C01827=1172.845,288.694,-69.686,-176.933,7.790,148.605
C01828=1172.841,288.942,-69.715,-176.930,7.793,148.605
C01829=1172.837,289.190,-69.744,-176.927,7.796,148.605
C01830=1172.832,289.439,-69.774,-176.925,7.799,148.605
C01831=1172.828,289.687,-69.805,-176.922,7.802,148.605
C01832=1172.824,289.935,-69.834,-176.920,7.805,148.605
C01833=1172.819,290.183,-69.864,-176.917,7.808,148.605
C01834=1172.815,290.431,-69.893,-176.914,7.811,148.605
C01835=1172.811,290.680,-69.923,-176.912,7.814,148.605
C01836=1172.807,290.928,-69.952,-176.910,7.816,148.605
C01837=1172.803,291.176,-69.981,-176.907,7.819,148.605
C01838=1172.798,291.424,-70.012,-176.904,7.822,148.605
C01839=1172.794,291.673,-70.042,-176.901,7.825,148.605
C01840=1172.790,291.921,-70.071,-176.899,7.828,148.605
C01841=1172.785,292.169,-70.101,-176.896,7.831,148.605
C01842=1172.781,292.417,-70.131,-176.894,7.834,148.605
C01843=1172.777,292.665,-70.161,-176.891,7.837,148.605
C01844=1172.772,292.914,-70.190,-176.889,7.841,148.605
C01845=1172.768,293.162,-70.220,-176.886,7.844,148.605
C01846=1172.764,293.409,-70.250,-176.883,7.847,148.605
C01847=1172.760,293.658,-70.280,-176.881,7.849,148.605
C01848=1172.755,293.906,-70.309,-176.878,7.852,148.605
C01849=1172.751,294.154,-70.339,-176.876,7.855,148.605
C01850=1172.747,294.403,-70.370,-176.873,7.858,148.605
C01851=1172.742,294.651,-70.399,-176.871,7.861,148.605
C01852=1172.738,294.898,-70.429,-176.868,7.864,148.605
C01853=1172.734,295.147,-70.459,-176.866,7.867,148.605
C01854=1172.730,295.395,-70.489,-176.863,7.870,148.605
C01855=1172.726,295.643,-70.519,-176.860,7.873,148.605
C01856=1172.721,295.891,-70.548,-176.857,7.876,148.605
C01857=1172.717,296.140,-70.579,-176.855,7.880,148.605
C01858=1172.713,296.388,-70.609,-176.852,7.883,148.605
C01859=1172.709,296.636,-70.640,-176.850,7.886,148.605
C01860=1172.704,296.884,-70.669,-176.847,7.888,148.605
C01861=1172.700,297.132,-70.699,-176.845,7.891,148.605
C01862=1172.696,297.381,-70.729,-176.842,7.894,148.605
C01863=1172.692,297.628,-70.759,-176.840,7.897,148.605
C01864=1172.687,297.876,-70.789,-176.837,7.900,148.605
C01865=1172.683,298.124,-70.820,-176.835,7.903,148.605
C01866=1172.679,298.373,-70.849,-176.832,7.906,148.605
C01867=1172.675,298.621,-70.880,-176.829,7.909,148.605
C01868=1172.671,298.869,-70.910,-176.827,7.912,148.606
C01869=1172.666,299.118,-70.940,-176.824,7.915,148.606
C01870=1172.662,299.365,-70.971,-176.821,7.918,148.606
C01871=1172.657,299.614,-71.001,-176.819,7.921,148.605
C01872=1172.653,299.861,-71.031,-176.816,7.925,148.606
C01873=1172.649,300.110,-71.062,-176.814,7.928,148.606
C01874=1172.645,300.358,-71.091,-176.811,7.931,148.606
C01875=1172.640,300.606,-71.122,-176.809,7.934,148.606
C01876=1172.637,300.854,-71.152,-176.806,7.937,148.606
C01877=1172.632,301.102,-71.183,-176.804,7.939,148.606
C01878=1172.628,301.350,-71.213,-176.801,7.942,148.606
C01879=1172.624,301.599,-71.244,-176.799,7.945,148.606
C01880=1172.620,301.847,-71.274,-176.796,7.948,148.606
C01881=1172.615,302.094,-71.305,-176.793,7.951,148.606
C01882=1172.611,302.343,-71.334,-176.791,7.955,148.606
C01883=1172.606,302.591,-71.365,-176.788,7.958,148.606
C01884=1172.602,302.839,-71.396,-176.786,7.961,148.606
C01885=1172.599,303.087,-71.426,-176.783,7.964,148.606
C01886=1172.594,303.335,-71.457,-176.781,7.967,148.606
C01887=1172.590,303.583,-71.486,-176.778,7.970,148.606
C01888=1172.586,303.832,-71.518,-176.776,7.973,148.606
C01889=1172.581,304.080,-71.548,-176.773,7.976,148.606
C01890=1172.577,304.328,-71.578,-176.770,7.979,148.606
C01891=1172.573,304.575,-71.609,-176.768,7.982,148.606
C01892=1172.568,304.823,-71.640,-176.765,7.985,148.606
C01893=1172.565,305.072,-71.671,-176.763,7.989,148.607
C01894=1172.560,305.320,-71.701,-176.760,7.992,148.607
C01895=1172.556,305.568,-71.732,-176.757,7.995,148.607
C01896=1172.552,305.816,-71.763,-176.755,7.998,148.607
C01897=1172.547,306.065,-71.793,-176.752,8.001,148.607
C01898=1172.543,306.313,-71.823,-176.750,8.004,148.607
C01899=1172.539,306.560,-71.854,-176.747,8.007,148.607
C01900=1172.535,306.809,-71.885,-176.745,8.010,148.607
C01901=1172.531,307.056,-71.916,-176.742,8.013,148.607
C01902=1172.526,307.304,-71.947,-176.739,8.017,148.607
C01903=1172.523,307.553,-71.977,-176.737,8.019,148.607
C01904=1172.518,307.800,-72.008,-176.734,8.023,148.607
C01905=1172.513,308.048,-72.039,-176.732,8.026,148.607
C01906=1172.509,308.297,-72.070,-176.729,8.029,148.607
C01907=1172.505,308.545,-72.101,-176.727,8.032,148.607
C01908=1172.501,308.793,-72.131,-176.724,8.035,148.607
C01909=1172.497,309.041,-72.162,-176.721,8.038,148.607
C01910=1172.492,309.289,-72.193,-176.719,8.041,148.608
C01911=1172.488,309.537,-72.224,-176.716,8.044,148.607
C01912=1172.484,309.785,-72.256,-176.714,8.048,148.608
C01913=1172.480,310.033,-72.286,-176.711,8.051,148.608
C01914=1172.475,310.281,-72.317,-176.709,8.054,148.608
C01915=1172.471,310.530,-72.348,-176.706,8.057,148.608
C01916=1172.467,310.777,-72.379,-176.704,8.060,148.608
C01917=1172.463,311.026,-72.410,-176.701,8.063,148.608
C01918=1172.459,311.274,-72.441,-176.698,8.066,148.608
C01919=1172.454,311.522,-72.472,-176.696,8.069,148.608
C01920=1172.451,311.769,-72.503,-176.693,8.072,148.608
C01921=1172.446,312.017,-72.534,-176.691,8.075,148.608
C01922=1172.442,312.266,-72.565,-176.688,8.079,148.608
C01923=1172.438,312.513,-72.596,-176.686,8.082,148.608
C01924=1172.433,312.761,-72.627,-176.683,8.085,148.609
C01925=1172.429,313.010,-72.658,-176.681,8.088,148.609
C01926=1172.425,313.257,-72.690,-176.678,8.091,148.609
C01927=1172.421,313.506,-72.721,-176.676,8.094,148.609
C01928=1172.416,313.783,-72.756,-176.673,8.097,148.609
C01929=1172.412,314.060,-72.790,-176.670,8.101,148.609
C01930=1172.407,314.337,-72.825,-176.667,8.104,148.609
C01931=1172.403,314.613,-72.860,-176.665,8.108,148.609
C01932=1172.398,314.861,-72.891,-176.662,8.111,148.609
C01933=1172.394,315.109,-72.923,-176.660,8.115,148.609
C01934=1172.390,315.357,-72.953,-176.657,8.118,148.609
C01935=1172.386,315.605,-72.985,-176.655,8.121,148.610
C01936=1172.381,315.853,-73.016,-176.652,8.124,148.609
C01937=1172.378,316.101,-73.048,-176.650,8.127,148.610
C01938=1172.373,316.349,-73.079,-176.647,8.130,148.610
C01939=1172.369,316.597,-73.111,-176.644,8.133,148.610
C01940=1172.364,316.845,-73.142,-176.642,8.137,148.610
C01941=1172.360,317.093,-73.174,-176.639,8.140,148.610
C01942=1172.356,317.341,-73.205,-176.637,8.143,148.610
C01943=1172.352,317.589,-73.236,-176.634,8.146,148.610
C01944=1172.348,317.837,-73.268,-176.632,8.149,148.610
C01945=1172.344,318.085,-73.300,-176.629,8.152,148.610
C01946=1172.340,318.333,-73.331,-176.627,8.155,148.610
C01947=1172.336,318.581,-73.362,-176.624,8.158,148.610
C01948=1172.332,318.829,-73.393,-176.622,8.162,148.611
C01949=1172.327,319.077,-73.425,-176.619,8.165,148.611
C01950=1172.323,319.325,-73.457,-176.617,8.168,148.611
C01951=1172.319,319.572,-73.489,-176.614,8.171,148.611
C01952=1172.315,319.821,-73.520,-176.612,8.174,148.611
C01953=1172.311,320.069,-73.552,-176.609,8.178,148.611
C01954=1172.306,320.316,-73.583,-176.606,8.181,148.611
C01955=1172.303,320.564,-73.615,-176.604,8.185,148.611
C01956=1172.297,320.813,-73.646,-176.601,8.188,148.611
C01957=1172.294,321.061,-73.678,-176.599,8.191,148.612
C01958=1172.290,321.309,-73.710,-176.596,8.194,148.612
C01959=1172.286,321.556,-73.742,-176.594,8.197,148.612
C01960=1172.282,321.804,-73.773,-176.591,8.200,148.612
C01961=1172.277,322.052,-73.805,-176.589,8.204,148.612
C01962=1172.273,322.301,-73.837,-176.587,8.207,148.612
C01963=1172.269,322.549,-73.868,-176.584,8.210,148.612
C01964=1172.265,322.796,-73.900,-176.582,8.213,148.612
C01965=1172.260,323.044,-73.932,-176.579,8.216,148.612
C01966=1172.257,323.292,-73.964,-176.577,8.219,148.613
C01967=1172.252,323.540,-73.996,-176.574,8.222,148.613
C01968=1172.248,323.788,-74.028,-176.572,8.226,148.613
C01969=1172.244,324.036,-74.060,-176.569,8.229,148.613
C01970=1172.240,324.283,-74.091,-176.566,8.233,148.613
C01971=1172.236,324.531,-74.123,-176.564,8.236,148.613
C01972=1172.232,324.780,-74.156,-176.561,8.239,148.613
C01973=1172.228,325.027,-74.187,-176.559,8.242,148.613
C01974=1172.224,325.275,-74.219,-176.556,8.246,148.614
C01975=1172.219,325.523,-74.251,-176.554,8.249,148.614
C01976=1172.215,325.771,-74.283,-176.551,8.252,148.614
C01977=1172.211,326.019,-74.315,-176.549,8.255,148.614
C01978=1172.207,326.267,-74.347,-176.546,8.258,148.614
C01979=1172.203,326.515,-74.379,-176.544,8.262,148.614
C01980=1172.198,326.763,-74.411,-176.541,8.265,148.614
C01981=1172.194,327.011,-74.443,-176.539,8.268,148.614
C01982=1172.190,327.259,-74.475,-176.537,8.271,148.615
C01983=1172.186,327.507,-74.507,-176.533,8.275,148.615
C01984=1172.182,327.754,-74.539,-176.531,8.278,148.615
C01985=1172.178,328.002,-74.572,-176.529,8.282,148.615
C01986=1172.174,328.250,-74.604,-176.526,8.285,148.615
C01987=1172.169,328.498,-74.636,-176.524,8.288,148.615
C01988=1172.165,328.746,-74.668,-176.522,8.291,148.615
C01989=1172.161,328.994,-74.701,-176.519,8.294,148.615
C01990=1172.158,329.242,-74.733,-176.517,8.297,148.616
C01991=1172.153,329.490,-74.765,-176.514,8.301,148.616
C01992=1172.149,329.738,-74.797,-176.512,8.304,148.616
C01993=1172.145,329.985,-74.830,-176.509,8.307,148.616
C01994=1172.141,330.233,-74.862,-176.506,8.311,148.616
C01995=1172.137,330.482,-74.894,-176.504,8.314,148.616
C01996=1172.132,330.729,-74.926,-176.501,8.317,148.616
C01997=1172.128,330.977,-74.959,-176.499,8.321,148.617
C01998=1172.124,331.225,-74.991,-176.496,8.324,148.617
C01999=1172.120,331.473,-75.023,-176.494,8.327,148.617
C02000=1172.116,331.721,-75.056,-176.492,8.330,148.617
C02001=1172.112,331.969,-75.088,-176.490,8.334,148.617
C02002=1172.107,332.216,-75.121,-176.487,8.337,148.617
C02003=1172.104,332.464,-75.153,-176.484,8.341,148.618
C02004=1172.099,332.712,-75.185,-176.482,8.344,148.618
C02005=1172.095,332.960,-75.218,-176.479,8.347,148.618
C02006=1172.091,333.208,-75.250,-176.477,8.350,148.618
C02007=1172.087,333.456,-75.283,-176.474,8.354,148.618
C02008=1172.082,333.703,-75.315,-176.472,8.357,148.618
C02009=1172.079,333.951,-75.348,-176.469,8.360,148.618
C02010=1172.074,334.199,-75.380,-176.467,8.363,148.619
C02011=1172.070,334.447,-75.413,-176.464,8.367,148.619
C02012=1172.067,334.695,-75.445,-176.462,8.371,148.619
C02013=1172.062,334.943,-75.478,-176.460,8.374,148.619
C02014=1172.058,335.191,-75.511,-176.457,8.377,148.619
C02015=1172.055,335.438,-75.543,-176.455,8.380,148.619
C02016=1172.050,335.686,-75.577,-176.452,8.384,148.620
C02017=1172.045,335.934,-75.609,-176.450,8.387,148.620
C02018=1172.042,336.181,-75.641,-176.447,8.390,148.620
C02019=1172.038,336.430,-75.674,-176.445,8.394,148.620
C02020=1172.033,336.677,-75.707,-176.442,8.397,148.620
C02021=1172.029,336.925,-75.740,-176.440,8.401,148.621
C02022=1172.026,337.173,-75.772,-176.438,8.404,148.621
C02023=1172.021,337.421,-75.805,-176.435,8.407,148.621
C02024=1172.017,337.669,-75.838,-176.433,8.410,148.621
C02025=1172.013,337.916,-75.871,-176.431,8.413,148.621
C02026=1172.009,338.165,-75.904,-176.428,8.418,148.621
C02027=1172.005,338.412,-75.936,-176.425,8.421,148.622
C02028=1172.001,338.660,-75.969,-176.423,8.424,148.622
C02029=1171.997,338.908,-76.002,-176.421,8.428,148.622
C02030=1171.993,339.156,-76.035,-176.418,8.430,148.622
C02031=1171.988,339.404,-76.068,-176.416,8.434,148.622
C02032=1171.984,339.682,-76.105,-176.413,8.438,148.622
C02033=1171.979,339.962,-76.142,-176.410,8.442,148.623
C02034=1171.975,340.241,-76.180,-176.408,8.445,148.623
C02035=1171.970,340.520,-76.216,-176.405,8.449,148.623
C02036=1171.966,340.768,-76.249,-176.403,8.453,148.623
C02037=1171.962,341.016,-76.282,-176.400,8.456,148.623
C02038=1171.958,341.264,-76.315,-176.398,8.459,148.624
C02039=1171.953,341.511,-76.348,-176.395,8.463,148.624
C02040=1171.949,341.759,-76.381,-176.393,8.466,148.624
C02041=1171.945,342.007,-76.415,-176.390,8.470,148.624
C02042=1171.941,342.255,-76.448,-176.388,8.473,148.625
C02043=1171.937,342.502,-76.481,-176.386,8.476,148.625
C02044=1171.933,342.750,-76.514,-176.383,8.480,148.625
C02045=1171.929,342.999,-76.548,-176.381,8.484,148.625
C02046=1171.925,343.246,-76.581,-176.378,8.487,148.625
C02047=1171.921,343.494,-76.614,-176.376,8.490,148.626
C02048=1171.917,343.742,-76.647,-176.374,8.494,148.626
C02049=1171.913,343.989,-76.680,-176.371,8.497,148.626
C02050=1171.909,344.237,-76.713,-176.369,8.501,148.626
C02051=1171.904,344.485,-76.747,-176.366,8.504,148.627
C02052=1171.900,344.733,-76.780,-176.364,8.508,148.627
C02053=1171.896,344.980,-76.813,-176.361,8.511,148.627
C02054=1171.892,345.228,-76.846,-176.359,8.514,148.627
C02055=1171.888,345.476,-76.879,-176.357,8.517,148.627
C02056=1171.884,345.723,-76.913,-176.354,8.521,148.627
C02057=1171.880,345.971,-76.946,-176.352,8.525,148.628
C02058=1171.876,346.219,-76.980,-176.350,8.528,148.628
C02059=1171.872,346.467,-77.013,-176.348,8.532,148.628
C02060=1171.868,346.715,-77.046,-176.345,8.535,148.629
C02061=1171.863,346.963,-77.080,-176.342,8.539,148.629
C02062=1171.859,347.210,-77.114,-176.340,8.542,148.629
C02063=1171.855,347.457,-77.147,-176.338,8.546,148.629
C02064=1171.851,347.705,-77.180,-176.336,8.549,148.629
C02065=1171.848,347.954,-77.213,-176.333,8.552,148.630
C02066=1171.844,348.201,-77.247,-176.330,8.556,148.630
C02067=1171.840,348.448,-77.281,-176.328,8.560,148.630
C02068=1171.835,348.696,-77.314,-176.326,8.563,148.630
C02069=1171.831,348.944,-77.348,-176.324,8.566,148.631
C02070=1171.827,349.191,-77.381,-176.321,8.570,148.631
C02071=1171.823,349.440,-77.415,-176.318,8.574,148.631
C02072=1171.819,349.687,-77.449,-176.316,8.577,148.631
C02073=1171.815,349.935,-77.482,-176.314,8.580,148.631
C02074=1171.810,350.183,-77.516,-176.312,8.584,148.632
C02075=1171.806,350.430,-77.549,-176.309,8.588,148.632
C02076=1171.803,350.678,-77.583,-176.307,8.591,148.632
C02077=1171.799,350.925,-77.617,-176.305,8.595,148.633
C02078=1171.794,351.173,-77.651,-176.302,8.598,148.633
C02079=1171.790,351.421,-77.684,-176.300,8.601,148.633
C02080=1171.786,351.668,-77.718,-176.297,8.605,148.633
C02081=1171.783,351.917,-77.751,-176.295,8.609,148.634
C02082=1171.778,352.164,-77.786,-176.293,8.612,148.634
C02083=1171.774,352.412,-77.819,-176.291,8.616,148.634
C02084=1171.770,352.659,-77.853,-176.288,8.620,148.634
C02085=1171.767,352.907,-77.886,-176.286,8.623,148.635
C02086=1171.762,353.155,-77.921,-176.284,8.627,148.635
C02087=1171.758,353.402,-77.954,-176.282,8.630,148.635
C02088=1171.754,353.650,-77.988,-176.279,8.634,148.636
C02089=1171.750,353.898,-78.022,-176.276,8.637,148.636
C02090=1171.746,354.145,-78.056,-176.274,8.641,148.636
C02091=1171.742,354.392,-78.090,-176.272,8.644,148.636
C02092=1171.738,354.641,-78.124,-176.269,8.648,148.637
C02093=1171.734,354.888,-78.157,-176.267,8.652,148.637
C02094=1171.730,355.136,-78.192,-176.265,8.655,148.637
C02095=1171.726,355.384,-78.225,-176.263,8.659,148.638
C02096=1171.722,355.631,-78.259,-176.260,8.663,148.638
C02097=1171.718,355.879,-78.294,-176.258,8.666,148.638
C02098=1171.714,356.126,-78.328,-176.256,8.669,148.638
C02099=1171.709,356.375,-78.362,-176.254,8.673,148.639
C02100=1171.706,356.622,-78.396,-176.251,8.677,148.639
C02101=1171.702,356.869,-78.430,-176.249,8.680,148.639
C02102=1171.698,357.117,-78.464,-176.247,8.684,148.640
C02103=1171.694,357.365,-78.498,-176.245,8.687,148.640
C02104=1171.690,357.613,-78.532,-176.242,8.691,148.640
C02105=1171.686,357.860,-78.566,-176.240,8.695,148.640
C02106=1171.681,358.107,-78.601,-176.238,8.698,148.641
C02107=1171.678,358.355,-78.635,-176.235,8.702,148.641
C02108=1171.673,358.603,-78.669,-176.233,8.706,148.641
C02109=1171.669,358.850,-78.703,-176.231,8.709,148.642
C02110=1171.665,359.098,-78.737,-176.229,8.713,148.642
C02111=1171.662,359.345,-78.771,-176.226,8.717,148.642
C02112=1171.658,359.594,-78.806,-176.224,8.720,148.643
C02113=1171.654,359.841,-78.840,-176.222,8.724,148.643
C02114=1171.649,360.088,-78.874,-176.219,8.727,148.643
C02115=1171.646,360.336,-78.909,-176.217,8.732,148.644
C02116=1171.641,360.583,-78.943,-176.215,8.735,148.644
C02117=1171.638,360.831,-78.977,-176.213,8.739,148.644
C02118=1171.634,361.079,-79.012,-176.211,8.742,148.645
C02119=1171.630,361.327,-79.047,-176.208,8.746,148.645
C02120=1171.626,361.574,-79.081,-176.206,8.750,148.645
C02121=1171.621,361.821,-79.115,-176.204,8.753,148.646
C02122=1171.618,362.069,-79.149,-176.202,8.757,148.646
C02123=1171.613,362.316,-79.184,-176.199,8.761,148.646
C02124=1171.609,362.565,-79.219,-176.198,8.765,148.647
C02125=1171.606,362.812,-79.252,-176.195,8.768,148.647
C02126=1171.602,363.060,-79.287,-176.193,8.772,148.647
C02127=1171.598,363.307,-79.321,-176.191,8.776,148.648
C02128=1171.594,363.555,-79.356,-176.189,8.779,148.648
C02129=1171.589,363.802,-79.390,-176.187,8.783,148.649
C02130=1171.586,364.050,-79.425,-176.185,8.787,148.649
C02131=1171.582,364.297,-79.460,-176.182,8.791,148.649
C02132=1171.578,364.545,-79.495,-176.180,8.794,148.650
C02133=1171.574,364.792,-79.529,-176.179,8.798,148.650
C02134=1171.570,365.040,-79.563,-176.177,8.801,148.651
C02135=1171.566,365.287,-79.599,-176.175,8.805,148.651
C02136=1171.561,365.570,-79.638,-176.172,8.809,148.651
C02137=1171.556,365.852,-79.677,-176.170,8.814,148.652
C02138=1171.552,366.134,-79.717,-176.167,8.818,148.652
C02139=1171.548,366.415,-79.756,-176.165,8.822,148.653
C02140=1171.544,366.664,-79.791,-176.163,8.826,148.653
C02141=1171.540,366.911,-79.826,-176.161,8.830,148.654
C02142=1171.536,367.159,-79.861,-176.159,8.833,148.654
C02143=1171.532,367.407,-79.895,-176.157,8.837,148.654
C02144=1171.528,367.653,-79.930,-176.156,8.841,148.655
C02145=1171.524,367.901,-79.965,-176.154,8.844,148.655
C02146=1171.520,368.149,-79.999,-176.152,8.848,148.656
C02147=1171.516,368.396,-80.035,-176.150,8.851,148.656
C02148=1171.511,368.644,-80.069,-176.149,8.855,148.657
C02149=1171.507,368.892,-80.104,-176.146,8.860,148.657
C02150=1171.505,369.139,-80.139,-176.144,8.863,148.658
C02151=1171.500,369.386,-80.174,-176.142,8.867,148.658
C02152=1171.496,369.634,-80.209,-176.141,8.871,148.659
C02153=1171.492,369.881,-80.244,-176.139,8.874,148.659
C02154=1171.488,370.129,-80.279,-176.137,8.878,148.660
C02155=1171.484,370.377,-80.314,-176.136,8.882,148.660
C02156=1171.480,370.624,-80.349,-176.134,8.885,148.660
C02157=1171.477,370.871,-80.383,-176.132,8.889,148.661
C02158=1171.472,371.118,-80.419,-176.130,8.893,148.661
C02159=1171.468,371.366,-80.453,-176.129,8.896,148.662
C02160=1171.465,371.614,-80.489,-176.127,8.900,148.663
C02161=1171.460,371.861,-80.523,-176.125,8.904,148.663
C02162=1171.456,372.109,-80.559,-176.124,8.908,148.664
C02163=1171.452,372.357,-80.594,-176.122,8.911,148.664
C02164=1171.448,372.604,-80.629,-176.121,8.915,148.665
C02165=1171.444,372.852,-80.664,-176.119,8.918,148.665
C02166=1171.441,373.099,-80.699,-176.118,8.922,148.666
C02167=1171.436,373.346,-80.735,-176.116,8.926,148.666
C02168=1171.432,373.594,-80.769,-176.115,8.930,148.667
C02169=1171.429,373.842,-80.805,-176.113,8.933,148.667
C02170=1171.424,374.089,-80.840,-176.111,8.937,148.668
C02171=1171.420,374.337,-80.875,-176.111,8.940,148.668
C02172=1171.417,374.584,-80.911,-176.109,8.944,148.669
C02173=1171.413,374.831,-80.946,-176.107,8.948,148.669
C02174=1171.409,375.079,-80.981,-176.106,8.952,148.670
C02175=1171.405,375.327,-81.016,-176.104,8.955,148.670
C02176=1171.401,375.573,-81.051,-176.103,8.958,148.671
C02177=1171.397,375.822,-81.086,-176.102,8.962,148.672
C02178=1171.393,376.069,-81.122,-176.100,8.966,148.672
C02179=1171.389,376.316,-81.157,-176.100,8.969,148.673
C02180=1171.385,376.563,-81.192,-176.098,8.973,148.674
C02181=1171.381,376.811,-81.227,-176.097,8.977,148.674
C02182=1171.377,377.059,-81.263,-176.095,8.980,148.675
C02183=1171.373,377.306,-81.298,-176.094,8.984,148.675
C02184=1171.370,377.553,-81.334,-176.093,8.988,148.676
C02185=1171.366,377.801,-81.369,-176.092,8.991,148.676
C02186=1171.361,378.048,-81.404,-176.090,8.995,148.677
C02187=1171.358,378.296,-81.439,-176.090,8.998,148.678
C02188=1171.353,378.543,-81.475,-176.088,9.002,148.678
C02189=1171.350,378.791,-81.511,-176.088,9.005,148.679
C02190=1171.345,379.038,-81.546,-176.086,9.009,148.680
C02191=1171.342,379.285,-81.581,-176.085,9.012,148.680
C02192=1171.338,379.533,-81.617,-176.084,9.016,148.681
C02193=1171.334,379.781,-81.652,-176.083,9.019,148.681
C02194=1171.330,380.028,-81.687,-176.082,9.023,148.682
C02195=1171.326,380.275,-81.723,-176.081,9.026,148.683
C02196=1171.322,380.523,-81.759,-176.081,9.029,148.683
C02197=1171.318,380.771,-81.794,-176.079,9.033,148.684
C02198=1171.314,381.018,-81.830,-176.078,9.036,148.685
C02199=1171.310,381.265,-81.865,-176.078,9.040,148.685
C02200=1171.306,381.512,-81.901,-176.076,9.044,148.686
C02201=1171.303,381.760,-81.936,-176.076,9.047,148.687
C02202=1171.298,382.008,-81.972,-176.075,9.050,148.687
C02203=1171.294,382.254,-82.007,-176.074,9.053,148.688
C02204=1171.290,382.502,-82.043,-176.073,9.058,148.689
C02205=1171.287,382.749,-82.079,-176.073,9.061,148.689
C02206=1171.283,382.997,-82.114,-176.072,9.064,148.690
C02207=1171.279,383.245,-82.150,-176.071,9.067,148.691
C02208=1171.274,383.492,-82.185,-176.071,9.070,148.691
C02209=1171.271,383.739,-82.221,-176.070,9.074,148.692
C02210=1171.267,383.987,-82.257,-176.069,9.078,148.693
C02211=1171.263,384.234,-82.293,-176.068,9.081,148.693
C02212=1171.259,384.482,-82.328,-176.068,9.084,148.694
C02213=1171.255,384.729,-82.364,-176.067,9.087,148.695
C02214=1171.251,384.976,-82.399,-176.067,9.091,148.696
C02215=1171.247,385.224,-82.435,-176.066,9.094,148.696
C02216=1171.243,385.471,-82.471,-176.065,9.097,148.697
C02217=1171.239,385.719,-82.506,-176.065,9.100,148.698
C02218=1171.236,385.966,-82.542,-176.065,9.103,148.698
C02219=1171.232,386.214,-82.579,-176.064,9.106,148.699
C02220=1171.227,386.460,-82.614,-176.064,9.110,148.700
C02221=1171.224,386.708,-82.649,-176.063,9.113,148.700
C02222=1171.220,386.955,-82.685,-176.063,9.116,148.701
C02223=1171.216,387.203,-82.721,-176.063,9.119,148.702
C02224=1171.212,387.451,-82.757,-176.062,9.122,148.703
C02225=1171.208,387.698,-82.792,-176.062,9.126,148.703
C02226=1171.203,387.945,-82.828,-176.061,9.129,148.704
C02227=1171.200,388.192,-82.864,-176.062,9.131,148.705
C02228=1171.196,388.440,-82.900,-176.061,9.135,148.705
C02229=1171.193,388.687,-82.935,-176.061,9.137,148.706
C02230=1171.188,388.935,-82.971,-176.060,9.141,148.707
C02231=1171.185,389.183,-83.007,-176.060,9.144,148.708
C02232=1171.181,389.429,-83.043,-176.060,9.146,148.708
C02233=1171.177,389.677,-83.079,-176.060,9.150,148.709
C02234=1171.173,389.924,-83.114,-176.060,9.152,148.710
C02235=1171.169,390.172,-83.150,-176.060,9.156,148.711
C02236=1171.165,390.419,-83.186,-176.060,9.158,148.711
C02237=1171.161,390.666,-83.222,-176.059,9.161,148.712
C02238=1171.158,390.914,-83.258,-176.059,9.164,148.713
C02239=1171.153,391.162,-83.294,-176.059,9.167,148.713
C02240=1171.148,391.447,-83.335,-176.059,9.170,148.714
C02241=1171.144,391.731,-83.376,-176.059,9.174,148.715
C02242=1171.140,392.016,-83.417,-176.059,9.177,148.716
C02243=1171.136,392.301,-83.459,-176.059,9.180,148.717
C02244=1171.131,392.548,-83.495,-176.059,9.183,148.718
C02245=1171.127,392.795,-83.531,-176.059,9.185,148.718
C02246=1171.124,393.042,-83.567,-176.059,9.188,148.719
C02247=1171.120,393.290,-83.603,-176.059,9.191,148.720
C02248=1171.116,393.538,-83.639,-176.059,9.194,148.720
C02249=1171.112,393.785,-83.675,-176.059,9.196,148.721
C02250=1171.108,394.032,-83.711,-176.059,9.199,148.722
C02251=1171.104,394.280,-83.747,-176.060,9.201,148.723
C02252=1171.100,394.527,-83.782,-176.060,9.204,148.723
C02253=1171.096,394.775,-83.819,-176.060,9.206,148.724
C02254=1171.093,395.022,-83.855,-176.060,9.209,148.725
C02255=1171.088,395.269,-83.890,-176.060,9.212,148.725
C02256=1171.084,395.516,-83.927,-176.060,9.215,148.726
C02257=1171.081,395.763,-83.962,-176.060,9.218,148.727
C02258=1171.076,396.011,-83.998,-176.060,9.220,148.728
C02259=1171.073,396.258,-84.035,-176.060,9.223,148.728
C02260=1171.068,396.506,-84.071,-176.061,9.224,148.729
C02261=1171.065,396.754,-84.106,-176.061,9.227,148.730
C02262=1171.061,397.000,-84.143,-176.061,9.230,148.730
C02263=1171.057,397.248,-84.179,-176.061,9.232,148.731
C02264=1171.053,397.496,-84.214,-176.062,9.235,148.732
C02265=1171.049,397.743,-84.251,-176.062,9.237,148.733
C02266=1171.046,397.990,-84.287,-176.062,9.240,148.733
C02267=1171.041,398.237,-84.322,-176.062,9.242,148.734
C02268=1171.037,398.484,-84.359,-176.063,9.244,148.735
C02269=1171.034,398.732,-84.394,-176.063,9.247,148.735
C02270=1171.030,398.979,-84.431,-176.063,9.249,148.736
C02271=1171.026,399.227,-84.467,-176.063,9.252,148.737
C02272=1171.021,399.474,-84.503,-176.063,9.254,148.737
C02273=1171.018,399.721,-84.539,-176.064,9.256,148.738
C02274=1171.014,399.969,-84.575,-176.064,9.258,148.739
C02275=1171.010,400.217,-84.611,-176.064,9.261,148.739
C02276=1171.006,400.464,-84.648,-176.064,9.264,148.740
C02277=1171.002,400.711,-84.683,-176.065,9.265,148.741
C02278=1170.999,400.958,-84.719,-176.065,9.268,148.741
C02279=1170.995,401.206,-84.756,-176.065,9.270,148.742
C02280=1170.991,401.453,-84.791,-176.066,9.272,148.743
C02281=1170.987,401.701,-84.828,-176.066,9.274,148.743
C02282=1170.983,401.948,-84.864,-176.066,9.277,148.744
C02283=1170.978,402.195,-84.900,-176.066,9.279,148.745
C02284=1170.975,402.442,-84.936,-176.067,9.281,148.745
C02285=1170.971,402.689,-84.972,-176.067,9.283,148.746
C02286=1170.967,402.937,-85.008,-176.067,9.286,148.747
C02287=1170.963,403.185,-85.044,-176.067,9.288,148.747
C02288=1170.959,403.432,-85.080,-176.068,9.290,148.748
C02289=1170.955,403.679,-85.117,-176.068,9.292,148.749
C02290=1170.951,403.926,-85.153,-176.069,9.294,148.749
C02291=1170.947,404.174,-85.189,-176.069,9.297,148.750
C02292=1170.944,404.421,-85.225,-176.069,9.298,148.751
C02293=1170.939,404.669,-85.261,-176.069,9.301,148.751
C02294=1170.936,404.916,-85.298,-176.070,9.302,148.752
C02295=1170.932,405.163,-85.333,-176.070,9.305,148.753
C02296=1170.928,405.411,-85.369,-176.070,9.306,148.753
C02297=1170.925,405.658,-85.406,-176.071,9.309,148.754
C02298=1170.920,405.906,-85.442,-176.071,9.311,148.754
C02299=1170.917,406.152,-85.478,-176.071,9.313,148.755
C02300=1170.912,406.400,-85.514,-176.072,9.315,148.756
C02301=1170.909,406.647,-85.550,-176.072,9.317,148.756
C02302=1170.905,406.895,-85.587,-176.073,9.319,148.757
C02303=1170.901,407.142,-85.623,-176.072,9.321,148.757
C02304=1170.897,407.390,-85.659,-176.073,9.323,148.758
C02305=1170.894,407.637,-85.695,-176.074,9.325,148.759
C02306=1170.889,407.884,-85.731,-176.073,9.327,148.759
C02307=1170.886,408.131,-85.768,-176.074,9.329,148.760
C02308=1170.881,408.379,-85.804,-176.074,9.331,148.761
C02309=1170.878,408.626,-85.840,-176.075,9.333,148.761
C02310=1170.874,408.874,-85.876,-176.075,9.334,148.762
C02311=1170.870,409.121,-85.912,-176.075,9.337,148.762
C02312=1170.865,409.368,-85.948,-176.076,9.338,148.763
C02313=1170.862,409.615,-85.984,-176.076,9.341,148.764
C02314=1170.857,409.862,-86.021,-176.076,9.342,148.764
C02315=1170.854,410.109,-86.057,-176.077,9.344,148.765
C02316=1170.850,410.357,-86.093,-176.077,9.346,148.765
C02317=1170.846,410.604,-86.129,-176.077,9.348,148.766
C02318=1170.842,410.852,-86.165,-176.078,9.350,148.766
C02319=1170.838,411.099,-86.202,-176.078,9.352,148.767
C02320=1170.834,411.346,-86.238,-176.078,9.354,148.768
C02321=1170.830,411.594,-86.275,-176.079,9.355,148.768
C02322=1170.826,411.841,-86.310,-176.079,9.358,148.769
C02323=1170.822,412.088,-86.347,-176.079,9.359,148.769
C02324=1170.819,412.336,-86.383,-176.080,9.361,148.770
C02325=1170.815,412.583,-86.419,-176.080,9.363,148.771
C02326=1170.811,412.831,-86.455,-176.080,9.365,148.771
C02327=1170.807,413.078,-86.492,-176.081,9.367,148.772
C02328=1170.803,413.325,-86.527,-176.080,9.369,148.772
C02329=1170.799,413.572,-86.564,-176.081,9.371,148.773
C02330=1170.796,413.819,-86.601,-176.081,9.372,148.773
C02331=1170.791,414.067,-86.637,-176.081,9.375,148.774
C02332=1170.787,414.314,-86.674,-176.082,9.376,148.774
C02333=1170.784,414.562,-86.709,-176.082,9.377,148.775
C02334=1170.779,414.809,-86.746,-176.082,9.380,148.776
C02335=1170.776,415.057,-86.782,-176.082,9.381,148.776
C02336=1170.772,415.304,-86.818,-176.083,9.383,148.777
C02337=1170.768,415.551,-86.854,-176.083,9.385,148.777
C02338=1170.766,415.798,-86.890,-176.083,9.387,148.778
C02339=1170.765,416.046,-86.926,-176.083,9.388,148.778
C02340=1170.764,416.328,-86.968,-176.084,9.390,148.779
C02341=1170.765,416.610,-87.008,-176.084,9.392,148.779
C02342=1170.767,416.890,-87.049,-176.085,9.394,148.780
C02343=1170.770,417.172,-87.089,-176.085,9.396,148.780
C02344=1170.349,417.173,-87.134,-176.088,9.407,148.784
C02345=1170.346,416.889,-87.093,-176.087,9.405,148.783
C02346=1170.344,416.605,-87.052,-176.087,9.403,148.783
C02347=1170.343,416.320,-87.011,-176.087,9.401,148.783
C02348=1170.344,416.034,-86.970,-176.087,9.399,148.782
C02349=1170.345,415.788,-86.933,-176.086,9.398,148.781
C02350=1170.348,415.540,-86.897,-176.086,9.395,148.781
C02351=1170.351,415.293,-86.861,-176.086,9.394,148.780
C02352=1170.355,415.046,-86.824,-176.086,9.392,148.780
C02353=1170.359,414.798,-86.789,-176.085,9.391,148.779
C02354=1170.363,414.551,-86.752,-176.085,9.388,148.779
C02355=1170.367,414.304,-86.716,-176.085,9.387,148.778
C02356=1170.371,414.056,-86.680,-176.084,9.385,148.778
C02357=1170.375,413.809,-86.643,-176.085,9.383,148.777
C02358=1170.378,413.562,-86.607,-176.084,9.381,148.776
C02359=1170.383,413.314,-86.570,-176.084,9.380,148.776
C02360=1170.386,413.067,-86.535,-176.083,9.377,148.775
C02361=1170.390,412.820,-86.498,-176.083,9.376,148.775
C02362=1170.394,412.572,-86.462,-176.082,9.374,148.774
C02363=1170.398,412.325,-86.425,-176.082,9.373,148.774
C02364=1170.402,412.078,-86.390,-176.082,9.370,148.773
C02365=1170.406,411.830,-86.353,-176.082,9.369,148.772
C02366=1170.409,411.583,-86.317,-176.081,9.367,148.772
C02367=1170.414,411.336,-86.281,-176.081,9.365,148.771
C02368=1170.417,411.088,-86.245,-176.081,9.363,148.771
C02369=1170.421,410.841,-86.208,-176.080,9.361,148.770
C02370=1170.426,410.593,-86.172,-176.080,9.359,148.769
C02371=1170.429,410.346,-86.136,-176.080,9.357,148.769
C02372=1170.433,410.098,-86.100,-176.079,9.356,148.768
C02373=1170.437,409.852,-86.063,-176.079,9.353,148.768
C02374=1170.441,409.604,-86.027,-176.079,9.352,148.767
C02375=1170.445,409.357,-85.991,-176.079,9.349,148.767
C02376=1170.449,409.110,-85.954,-176.078,9.348,148.766
C02377=1170.452,408.862,-85.919,-176.078,9.346,148.765
C02378=1170.456,408.615,-85.882,-176.078,9.344,148.765
C02379=1170.460,408.368,-85.846,-176.077,9.342,148.764
C02380=1170.464,408.120,-85.809,-176.076,9.340,148.764
C02381=1170.468,407.873,-85.774,-176.077,9.338,148.763
C02382=1170.472,407.626,-85.737,-176.076,9.336,148.762
C02383=1170.476,407.378,-85.701,-176.076,9.334,148.762
C02384=1170.480,407.131,-85.665,-176.076,9.332,148.761
C02385=1170.483,406.883,-85.629,-176.075,9.330,148.761
C02386=1170.488,406.636,-85.593,-176.075,9.328,148.760
C02387=1170.491,406.389,-85.557,-176.074,9.326,148.759
C02388=1170.496,406.141,-85.520,-176.074,9.324,148.759
C02389=1170.499,405.894,-85.484,-176.074,9.322,148.758
C02390=1170.503,405.646,-85.448,-176.073,9.320,148.757
C02391=1170.507,405.399,-85.412,-176.073,9.318,148.757
C02392=1170.511,405.152,-85.376,-176.073,9.316,148.756
C02393=1170.514,404.905,-85.339,-176.072,9.314,148.756
C02394=1170.519,404.657,-85.303,-176.072,9.311,148.755
C02395=1170.522,404.410,-85.267,-176.071,9.309,148.754
C02396=1170.527,404.162,-85.231,-176.072,9.307,148.754
C02397=1170.530,403.915,-85.195,-176.071,9.305,148.753
C02398=1170.534,403.667,-85.158,-176.071,9.303,148.752
C02399=1170.538,403.421,-85.122,-176.070,9.301,148.752
C02400=1170.542,403.173,-85.086,-176.070,9.299,148.751
C02401=1170.546,402.926,-85.051,-176.070,9.297,148.750
C02402=1170.550,402.679,-85.014,-176.070,9.295,148.750
C02403=1170.554,402.431,-84.978,-176.069,9.292,148.749
C02404=1170.557,402.184,-84.942,-176.069,9.290,148.748
C02405=1170.562,401.937,-84.906,-176.069,9.288,148.748
C02406=1170.565,401.690,-84.870,-176.068,9.286,148.747
C02407=1170.570,401.442,-84.834,-176.068,9.283,148.746
C02408=1170.573,401.194,-84.798,-176.068,9.281,148.746
C02409=1170.577,400.947,-84.761,-176.067,9.279,148.745
C02410=1170.581,400.700,-84.726,-176.067,9.277,148.744
C02411=1170.585,400.453,-84.689,-176.067,9.274,148.744
C02412=1170.589,400.205,-84.653,-176.066,9.273,148.743
C02413=1170.593,399.958,-84.616,-176.066,9.270,148.742
C02414=1170.597,399.710,-84.581,-176.066,9.267,148.742
C02415=1170.601,399.463,-84.545,-176.066,9.265,148.741
C02416=1170.604,399.216,-84.508,-176.065,9.263,148.740
C02417=1170.608,398.968,-84.473,-176.065,9.260,148.740
C02418=1170.612,398.720,-84.437,-176.065,9.258,148.739
C02419=1170.616,398.473,-84.400,-176.065,9.255,148.738
C02420=1170.621,398.226,-84.365,-176.064,9.253,148.737
C02421=1170.624,397.980,-84.328,-176.064,9.251,148.737
C02422=1170.629,397.732,-84.292,-176.064,9.248,148.736
C02423=1170.632,397.484,-84.257,-176.063,9.246,148.735
C02424=1170.636,397.237,-84.220,-176.063,9.243,148.735
C02425=1170.640,396.989,-84.184,-176.063,9.241,148.734
C02426=1170.644,396.742,-84.149,-176.063,9.238,148.733
C02427=1170.648,396.495,-84.112,-176.063,9.236,148.732
C02428=1170.651,396.247,-84.076,-176.063,9.233,148.732
C02429=1170.656,395.999,-84.040,-176.063,9.231,148.731
C02430=1170.659,395.753,-84.004,-176.062,9.228,148.730
C02431=1170.663,395.505,-83.968,-176.062,9.225,148.730
C02432=1170.667,395.257,-83.932,-176.062,9.223,148.729
C02433=1170.671,395.011,-83.896,-176.062,9.220,148.728
C02434=1170.676,394.763,-83.860,-176.062,9.218,148.727
C02435=1170.679,394.516,-83.825,-176.062,9.215,148.727
C02436=1170.683,394.269,-83.788,-176.062,9.213,148.726
C02437=1170.687,394.021,-83.752,-176.061,9.210,148.725
C02438=1170.691,393.774,-83.717,-176.061,9.207,148.725
C02439=1170.695,393.526,-83.680,-176.061,9.205,148.724
C02440=1170.698,393.279,-83.644,-176.061,9.202,148.723
C02441=1170.702,393.031,-83.609,-176.061,9.200,148.722
C02442=1170.706,392.784,-83.572,-176.061,9.196,148.722
C02443=1170.710,392.537,-83.536,-176.061,9.194,148.721
C02444=1170.714,392.289,-83.500,-176.061,9.191,148.720
C02445=1170.718,392.005,-83.459,-176.061,9.188,148.719
C02446=1170.723,391.720,-83.418,-176.061,9.185,148.719
C02447=1170.727,391.435,-83.376,-176.061,9.182,148.718
C02448=1170.732,391.150,-83.335,-176.061,9.178,148.717
C02449=1170.736,390.903,-83.300,-176.061,9.175,148.716
C02450=1170.740,390.655,-83.264,-176.061,9.172,148.715
C02451=1170.744,390.408,-83.227,-176.061,9.169,148.715
C02452=1170.747,390.161,-83.192,-176.061,9.167,148.714
C02453=1170.752,389.913,-83.156,-176.062,9.164,148.713
C02454=1170.755,389.665,-83.120,-176.062,9.161,148.713
C02455=1170.759,389.418,-83.084,-176.062,9.158,148.712
C02456=1170.764,389.171,-83.048,-176.062,9.155,148.711
C02457=1170.767,388.924,-83.013,-176.062,9.152,148.710
C02458=1170.771,388.676,-82.977,-176.062,9.149,148.710
C02459=1170.776,388.429,-82.941,-176.063,9.146,148.709
C02460=1170.779,388.182,-82.905,-176.063,9.142,148.708
C02461=1170.783,387.934,-82.869,-176.063,9.140,148.707
C02462=1170.787,387.686,-82.833,-176.064,9.137,148.707
C02463=1170.791,387.439,-82.797,-176.064,9.133,148.706
C02464=1170.795,387.192,-82.762,-176.064,9.131,148.705
C02465=1170.799,386.945,-82.727,-176.064,9.127,148.705
C02466=1170.803,386.697,-82.690,-176.065,9.124,148.704
C02467=1170.806,386.450,-82.654,-176.066,9.121,148.703
C02468=1170.810,386.202,-82.619,-176.066,9.117,148.702
C02469=1170.814,385.955,-82.582,-176.067,9.114,148.702
C02470=1170.819,385.708,-82.547,-176.066,9.112,148.701
C02471=1170.822,385.460,-82.512,-176.067,9.108,148.700
C02472=1170.826,385.213,-82.476,-176.068,9.105,148.700
C02473=1170.830,384.965,-82.440,-176.068,9.102,148.699
C02474=1170.834,384.717,-82.405,-176.069,9.099,148.698
C02475=1170.837,384.471,-82.368,-176.069,9.095,148.697
C02476=1170.842,384.224,-82.333,-176.070,9.092,148.697
C02477=1170.846,383.976,-82.297,-176.071,9.089,148.696
C02478=1170.850,383.728,-82.261,-176.071,9.085,148.695
C02479=1170.853,383.481,-82.226,-176.072,9.081,148.695
C02480=1170.857,383.233,-82.190,-176.073,9.078,148.694
C02481=1170.861,382.986,-82.155,-176.074,9.075,148.693
C02482=1170.866,382.739,-82.119,-176.074,9.072,148.693
C02483=1170.869,382.491,-82.083,-176.075,9.068,148.692
C02484=1170.873,382.244,-82.048,-176.076,9.065,148.691
C02485=1170.877,381.996,-82.012,-176.077,9.061,148.691
C02486=1170.881,381.749,-81.976,-176.078,9.058,148.690
C02487=1170.885,381.502,-81.941,-176.078,9.055,148.689
C02488=1170.889,381.254,-81.905,-176.079,9.051,148.689
C02489=1170.893,381.007,-81.870,-176.080,9.048,148.688
C02490=1170.896,380.759,-81.834,-176.081,9.044,148.687
C02491=1170.901,380.512,-81.799,-176.082,9.040,148.687
C02492=1170.905,380.265,-81.763,-176.083,9.037,148.686
C02493=1170.909,380.017,-81.728,-176.084,9.034,148.685
C02494=1170.913,379.769,-81.693,-176.085,9.030,148.685
C02495=1170.916,379.522,-81.657,-176.086,9.027,148.684
C02496=1170.921,379.275,-81.622,-176.087,9.023,148.683
C02497=1170.924,379.027,-81.586,-176.088,9.020,148.683
C02498=1170.928,378.780,-81.551,-176.089,9.016,148.682
C02499=1170.932,378.532,-81.515,-176.090,9.013,148.682
C02500=1170.937,378.285,-81.479,-176.092,9.009,148.681
C02501=1170.940,378.037,-81.445,-176.092,9.006,148.680
C02502=1170.944,377.789,-81.409,-176.094,9.002,148.680
C02503=1170.948,377.543,-81.374,-176.095,8.998,148.679
C02504=1170.952,377.295,-81.338,-176.096,8.995,148.679
C02505=1170.956,377.048,-81.303,-176.097,8.991,148.678
C02506=1170.960,376.800,-81.268,-176.098,8.988,148.677
C02507=1170.964,376.553,-81.233,-176.100,8.984,148.677
C02508=1170.968,376.305,-81.197,-176.101,8.980,148.676
C02509=1170.971,376.058,-81.162,-176.103,8.976,148.676
C02510=1170.975,375.810,-81.126,-176.103,8.973,148.675
C02511=1170.980,375.563,-81.091,-176.105,8.969,148.674
C02512=1170.984,375.315,-81.056,-176.107,8.966,148.674
C02513=1170.988,375.068,-81.020,-176.107,8.963,148.673
C02514=1170.992,374.820,-80.986,-176.109,8.959,148.673
C02515=1170.996,374.573,-80.950,-176.110,8.955,148.672
C02516=1170.999,374.325,-80.914,-176.112,8.951,148.672
C02517=1171.004,374.078,-80.880,-176.114,8.947,148.671
C02518=1171.008,373.830,-80.844,-176.115,8.943,148.670
C02519=1171.011,373.583,-80.809,-176.116,8.940,148.670
C02520=1171.016,373.335,-80.774,-176.118,8.937,148.669
C02521=1171.020,373.088,-80.739,-176.120,8.933,148.669
C02522=1171.023,372.841,-80.704,-176.121,8.929,148.668
C02523=1171.027,372.593,-80.669,-176.123,8.925,148.668
C02524=1171.031,372.346,-80.634,-176.124,8.922,148.667
C02525=1171.035,372.098,-80.599,-176.126,8.918,148.667
C02526=1171.039,371.851,-80.564,-176.127,8.914,148.666
C02527=1171.043,371.603,-80.528,-176.129,8.910,148.666
C02528=1171.047,371.355,-80.494,-176.131,8.907,148.665
C02529=1171.051,371.108,-80.458,-176.133,8.903,148.665
C02530=1171.055,370.860,-80.424,-176.134,8.899,148.664
C02531=1171.059,370.613,-80.388,-176.136,8.895,148.664
C02532=1171.063,370.365,-80.353,-176.138,8.892,148.663
C02533=1171.067,370.118,-80.318,-176.140,8.888,148.663
C02534=1171.071,369.871,-80.284,-176.141,8.885,148.662
C02535=1171.074,369.623,-80.249,-176.143,8.881,148.662
C02536=1171.078,369.375,-80.214,-176.145,8.877,148.661
C02537=1171.083,369.128,-80.179,-176.146,8.873,148.661
C02538=1171.086,368.880,-80.144,-176.148,8.870,148.660
C02539=1171.091,368.633,-80.109,-176.150,8.866,148.660
C02540=1171.095,368.385,-80.074,-176.152,8.863,148.660
C02541=1171.099,368.138,-80.040,-176.154,8.859,148.659
C02542=1171.103,367.890,-80.005,-176.156,8.855,148.659
C02543=1171.106,367.642,-79.969,-176.158,8.851,148.658
C02544=1171.111,367.395,-79.935,-176.160,8.847,148.658
C02545=1171.115,367.147,-79.900,-176.162,8.844,148.657
C02546=1171.118,366.900,-79.866,-176.164,8.840,148.657
C02547=1171.122,366.652,-79.831,-176.165,8.837,148.657
C02548=1171.127,366.405,-79.796,-176.167,8.833,148.656
C02549=1171.131,366.123,-79.756,-176.170,8.828,148.656
C02550=1171.136,365.841,-79.717,-176.172,8.824,148.655
C02551=1171.140,365.559,-79.677,-176.175,8.820,148.655
C02552=1171.144,365.276,-79.637,-176.176,8.816,148.654
C02553=1171.148,365.029,-79.603,-176.179,8.812,148.654
C02554=1171.152,364.781,-79.569,-176.181,8.808,148.653
C02555=1171.157,364.534,-79.533,-176.183,8.804,148.653
C02556=1171.160,364.286,-79.499,-176.185,8.801,148.653
C02557=1171.164,364.039,-79.465,-176.187,8.797,148.652
C02558=1171.168,363.791,-79.430,-176.189,8.793,148.652
C02559=1171.172,363.544,-79.396,-176.191,8.790,148.652
C02560=1171.176,363.296,-79.361,-176.193,8.786,148.651
C02561=1171.180,363.049,-79.326,-176.195,8.783,148.651
C02562=1171.184,362.801,-79.292,-176.198,8.778,148.650
C02563=1171.188,362.554,-79.257,-176.200,8.775,148.650
C02564=1171.192,362.305,-79.222,-176.202,8.771,148.650
C02565=1171.196,362.058,-79.189,-176.204,8.768,148.649
C02566=1171.201,361.811,-79.154,-176.206,8.763,148.649
C02567=1171.205,361.563,-79.119,-176.209,8.760,148.649
C02568=1171.208,361.316,-79.085,-176.210,8.757,148.648
C02569=1171.212,361.068,-79.051,-176.213,8.752,148.648
C02570=1171.216,360.820,-79.017,-176.215,8.749,148.648
C02571=1171.220,360.572,-78.982,-176.217,8.746,148.647
C02572=1171.224,360.325,-78.948,-176.219,8.742,148.647
C02573=1171.228,360.077,-78.913,-176.222,8.738,148.647
C02574=1171.232,359.830,-78.879,-176.224,8.734,148.646
C02575=1171.236,359.583,-78.845,-176.226,8.731,148.646
C02576=1171.240,359.334,-78.810,-176.229,8.728,148.646
C02577=1171.244,359.087,-78.776,-176.231,8.723,148.645
C02578=1171.248,358.839,-78.742,-176.233,8.720,148.645
C02579=1171.252,358.592,-78.708,-176.235,8.716,148.645
C02580=1171.257,358.344,-78.674,-176.238,8.712,148.644
C02581=1171.260,358.096,-78.639,-176.240,8.709,148.644
C02582=1171.265,357.849,-78.605,-176.242,8.705,148.644
C02583=1171.268,357.602,-78.571,-176.244,8.702,148.644
C02584=1171.272,357.354,-78.537,-176.247,8.698,148.643
C02585=1171.277,357.106,-78.503,-176.249,8.694,148.643
C02586=1171.280,356.858,-78.469,-176.251,8.691,148.643
C02587=1171.284,356.611,-78.434,-176.254,8.687,148.642
C02588=1171.288,356.364,-78.401,-176.256,8.683,148.642
C02589=1171.292,356.115,-78.366,-176.258,8.680,148.642
C02590=1171.296,355.868,-78.333,-176.261,8.677,148.641
C02591=1171.300,355.621,-78.299,-176.263,8.672,148.641
C02592=1171.304,355.372,-78.265,-176.265,8.669,148.641
C02593=1171.308,355.125,-78.231,-176.268,8.665,148.641
C02594=1171.313,354.877,-78.196,-176.270,8.662,148.640
C02595=1171.317,354.630,-78.163,-176.272,8.658,148.640
C02596=1171.320,354.382,-78.129,-176.275,8.654,148.640
C02597=1171.325,354.134,-78.094,-176.277,8.651,148.639
C02598=1171.329,353.887,-78.061,-176.279,8.648,148.639
C02599=1171.332,353.639,-78.027,-176.281,8.643,148.639
C02600=1171.337,353.391,-77.993,-176.284,8.640,148.639
C02601=1171.341,353.144,-77.959,-176.286,8.637,148.638
C02602=1171.345,352.897,-77.926,-176.288,8.634,148.638
C02603=1171.349,352.648,-77.891,-176.291,8.629,148.638
C02604=1171.353,352.401,-77.858,-176.293,8.626,148.637
C02605=1171.357,352.153,-77.824,-176.295,8.622,148.637
C02606=1171.361,351.906,-77.790,-176.298,8.619,148.637
C02607=1171.365,351.657,-77.756,-176.300,8.615,148.637
C02608=1171.369,351.410,-77.722,-176.303,8.612,148.636
C02609=1171.373,351.162,-77.689,-176.305,8.608,148.636
C02610=1171.378,350.915,-77.655,-176.307,8.605,148.636
C02611=1171.381,350.666,-77.621,-176.310,8.601,148.636
C02612=1171.385,350.419,-77.588,-176.312,8.597,148.635
C02613=1171.389,350.172,-77.554,-176.314,8.594,148.635
C02614=1171.394,349.924,-77.521,-176.317,8.591,148.635
C02615=1171.398,349.676,-77.487,-176.319,8.588,148.635
C02616=1171.401,349.428,-77.453,-176.322,8.583,148.634
C02617=1171.405,349.180,-77.420,-176.324,8.580,148.634
C02618=1171.409,348.933,-77.386,-176.326,8.577,148.634
C02619=1171.414,348.685,-77.352,-176.329,8.573,148.634
C02620=1171.418,348.437,-77.319,-176.331,8.569,148.633
C02621=1171.422,348.190,-77.285,-176.333,8.566,148.633
C02622=1171.426,347.942,-77.252,-176.336,8.562,148.633
C02623=1171.430,347.694,-77.219,-176.338,8.559,148.633
C02624=1171.434,347.446,-77.186,-176.340,8.556,148.632
C02625=1171.438,347.199,-77.152,-176.343,8.552,148.632
C02626=1171.443,346.951,-77.118,-176.345,8.548,148.632
C02627=1171.447,346.704,-77.085,-176.347,8.545,148.632
C02628=1171.451,346.456,-77.052,-176.350,8.542,148.632
C02629=1171.454,346.208,-77.017,-176.352,8.539,148.631
C02630=1171.458,345.960,-76.984,-176.355,8.534,148.631
C02631=1171.462,345.713,-76.951,-176.357,8.531,148.631
C02632=1171.467,345.465,-76.918,-176.359,8.528,148.631
C02633=1171.471,345.217,-76.885,-176.362,8.524,148.630
C02634=1171.475,344.969,-76.852,-176.364,8.521,148.630
C02635=1171.479,344.722,-76.818,-176.367,8.517,148.630
C02636=1171.483,344.474,-76.785,-176.369,8.514,148.630
C02637=1171.487,344.227,-76.751,-176.371,8.510,148.630
C02638=1171.491,343.979,-76.718,-176.374,8.507,148.629
C02639=1171.495,343.731,-76.685,-176.376,8.504,148.629
C02640=1171.499,343.483,-76.652,-176.378,8.501,148.629
C02641=1171.503,343.235,-76.618,-176.381,8.496,148.629
C02642=1171.507,342.987,-76.585,-176.383,8.493,148.628
C02643=1171.511,342.740,-76.552,-176.386,8.490,148.628
C02644=1171.515,342.492,-76.519,-176.388,8.487,148.628
C02645=1171.519,342.244,-76.486,-176.391,8.484,148.628
C02646=1171.524,341.997,-76.453,-176.394,8.479,148.628
C02647=1171.528,341.749,-76.419,-176.396,8.476,148.628
C02648=1171.532,341.500,-76.387,-176.398,8.473,148.627
C02649=1171.536,341.253,-76.354,-176.400,8.470,148.627
C02650=1171.540,341.005,-76.321,-176.403,8.466,148.627
C02651=1171.545,340.757,-76.288,-176.405,8.463,148.627
C02652=1171.549,340.510,-76.254,-176.408,8.459,148.626
C02653=1171.553,340.230,-76.217,-176.410,8.456,148.626
C02654=1171.558,339.951,-76.180,-176.413,8.451,148.626
C02655=1171.562,339.672,-76.143,-176.416,8.448,148.626
C02656=1171.567,339.392,-76.105,-176.419,8.444,148.626
C02657=1171.571,339.144,-76.073,-176.421,8.440,148.625
C02658=1171.575,338.896,-76.040,-176.424,8.437,148.625
C02659=1171.579,338.649,-76.007,-176.426,8.434,148.625
C02660=1171.583,338.401,-75.974,-176.428,8.430,148.625
C02661=1171.588,338.153,-75.942,-176.431,8.427,148.625
C02662=1171.592,337.906,-75.909,-176.433,8.424,148.625
C02663=1171.596,337.658,-75.876,-176.436,8.421,148.624
C02664=1171.600,337.411,-75.843,-176.438,8.417,148.624
C02665=1171.604,337.162,-75.811,-176.441,8.413,148.624
C02666=1171.608,336.914,-75.777,-176.443,8.410,148.624
C02667=1171.612,336.667,-75.745,-176.446,8.407,148.624
C02668=1171.616,336.419,-75.712,-176.448,8.404,148.624
C02669=1171.620,336.171,-75.679,-176.450,8.400,148.623
C02670=1171.624,335.923,-75.646,-176.453,8.397,148.623
C02671=1171.628,335.675,-75.614,-176.455,8.393,148.623
C02672=1171.632,335.427,-75.581,-176.458,8.390,148.623
C02673=1171.637,335.179,-75.549,-176.460,8.387,148.623
C02674=1171.640,334.932,-75.516,-176.463,8.383,148.622
C02675=1171.645,334.684,-75.484,-176.465,8.380,148.622
C02676=1171.649,334.436,-75.451,-176.467,8.377,148.622
C02677=1171.653,334.189,-75.418,-176.470,8.374,148.622
C02678=1171.657,333.941,-75.386,-176.472,8.370,148.622
C02679=1171.661,333.693,-75.353,-176.475,8.366,148.622
C02680=1171.665,333.445,-75.321,-176.477,8.363,148.621
C02681=1171.670,333.196,-75.288,-176.480,8.360,148.621
C02682=1171.674,332.949,-75.255,-176.482,8.357,148.621
C02683=1171.678,332.701,-75.224,-176.485,8.353,148.621
C02684=1171.682,332.454,-75.191,-176.487,8.350,148.621
C02685=1171.687,332.205,-75.158,-176.490,8.347,148.621
C02686=1171.690,331.958,-75.126,-176.492,8.344,148.621
C02687=1171.694,331.709,-75.093,-176.495,8.340,148.620
C02688=1171.698,331.461,-75.061,-176.498,8.337,148.620
C02689=1171.703,331.214,-75.029,-176.500,8.333,148.620
C02690=1171.707,330.966,-74.997,-176.502,8.330,148.620
C02691=1171.711,330.718,-74.964,-176.504,8.327,148.620
C02692=1171.715,330.470,-74.931,-176.507,8.324,148.620
C02693=1171.719,330.222,-74.899,-176.509,8.321,148.619
C02694=1171.724,329.975,-74.867,-176.512,8.317,148.619
C02695=1171.727,329.727,-74.835,-176.514,8.314,148.619
C02696=1171.732,329.479,-74.802,-176.517,8.310,148.619
C02697=1171.735,329.231,-74.770,-176.520,8.307,148.619
C02698=1171.740,328.983,-74.738,-176.522,8.304,148.619
C02699=1171.744,328.736,-74.706,-176.525,8.301,148.619
C02700=1171.748,328.487,-74.673,-176.527,8.297,148.618
C02701=1171.752,328.239,-74.641,-176.530,8.294,148.618
C02702=1171.756,327.991,-74.609,-176.532,8.291,148.618
C02703=1171.761,327.744,-74.578,-176.534,8.288,148.618
C02704=1171.764,327.496,-74.545,-176.537,8.285,148.618
C02705=1171.769,327.248,-74.513,-176.539,8.281,148.618
C02706=1171.773,327.001,-74.481,-176.542,8.277,148.618
C02707=1171.777,326.752,-74.449,-176.545,8.274,148.618
C02708=1171.781,326.504,-74.417,-176.547,8.271,148.617
C02709=1171.786,326.256,-74.384,-176.549,8.268,148.617
C02710=1171.790,326.008,-74.353,-176.552,8.265,148.617
C02711=1171.794,325.760,-74.321,-176.554,8.261,148.617
C02712=1171.798,325.512,-74.289,-176.557,8.258,148.617
C02713=1171.802,325.265,-74.257,-176.559,8.255,148.617
C02714=1171.806,325.017,-74.225,-176.562,8.252,148.617
C02715=1171.810,324.769,-74.192,-176.564,8.249,148.617
C02716=1171.814,324.521,-74.160,-176.567,8.245,148.616
C02717=1171.818,324.273,-74.129,-176.569,8.243,148.616
C02718=1171.823,324.025,-74.097,-176.572,8.238,148.616
C02719=1171.827,323.777,-74.065,-176.574,8.235,148.616
C02720=1171.831,323.529,-74.034,-176.577,8.232,148.616
C02721=1171.835,323.281,-74.001,-176.579,8.229,148.616
C02722=1171.839,323.033,-73.969,-176.582,8.226,148.616
C02723=1171.843,322.786,-73.938,-176.584,8.223,148.616
C02724=1171.847,322.538,-73.906,-176.587,8.219,148.615
C02725=1171.852,322.290,-73.874,-176.589,8.216,148.615
C02726=1171.856,322.042,-73.842,-176.592,8.213,148.615
C02727=1171.860,321.794,-73.810,-176.594,8.210,148.615
C02728=1171.864,321.546,-73.780,-176.597,8.207,148.615
C02729=1171.869,321.297,-73.747,-176.599,8.204,148.615
C02730=1171.872,321.049,-73.715,-176.602,8.200,148.615
C02731=1171.877,320.802,-73.684,-176.604,8.197,148.615
C02732=1171.880,320.554,-73.652,-176.607,8.194,148.615
C02733=1171.885,320.306,-73.621,-176.609,8.191,148.614
C02734=1171.889,320.058,-73.589,-176.612,8.187,148.614
C02735=1171.893,319.810,-73.557,-176.615,8.184,148.614
C02736=1171.897,319.562,-73.525,-176.617,8.181,148.614
C02737=1171.901,319.314,-73.494,-176.620,8.177,148.614
C02738=1171.906,319.066,-73.463,-176.622,8.174,148.614
C02739=1171.909,318.818,-73.431,-176.625,8.171,148.614
C02740=1171.914,318.571,-73.399,-176.627,8.168,148.614
C02741=1171.918,318.322,-73.368,-176.630,8.165,148.614
C02742=1171.922,318.074,-73.336,-176.632,8.162,148.614
C02743=1171.927,317.826,-73.305,-176.635,8.159,148.613
C02744=1171.930,317.578,-73.273,-176.637,8.156,148.613
C02745=1171.935,317.331,-73.242,-176.640,8.152,148.613
C02746=1171.939,317.082,-73.211,-176.642,8.149,148.613
C02747=1171.943,316.835,-73.179,-176.645,8.146,148.613
C02748=1171.947,316.586,-73.148,-176.647,8.143,148.613
C02749=1171.951,316.339,-73.117,-176.650,8.140,148.613
C02750=1171.955,316.091,-73.085,-176.652,8.137,148.613
C02751=1171.960,315.843,-73.054,-176.655,8.133,148.613
C02752=1171.963,315.595,-73.022,-176.657,8.130,148.613
C02753=1171.968,315.347,-72.991,-176.660,8.127,148.613
C02754=1171.972,315.099,-72.960,-176.662,8.124,148.613
C02755=1171.976,314.851,-72.929,-176.665,8.121,148.612
C02756=1171.980,314.602,-72.898,-176.667,8.118,148.612
C02757=1171.985,314.325,-72.862,-176.670,8.114,148.612
C02758=1171.990,314.048,-72.827,-176.673,8.111,148.612
C02759=1171.994,313.772,-72.793,-176.676,8.107,148.612
C02760=1172.000,313.494,-72.758,-176.679,8.104,148.612
C02761=1172.004,313.247,-72.727,-176.681,8.101,148.612
C02762=1172.008,312.998,-72.695,-176.684,8.097,148.612
C02763=1172.012,312.751,-72.664,-176.686,8.094,148.612
C02764=1172.016,312.502,-72.633,-176.689,8.090,148.612
C02765=1172.021,312.254,-72.602,-176.692,8.087,148.612
C02766=1172.024,312.007,-72.571,-176.694,8.084,148.611
C02767=1172.028,311.759,-72.540,-176.697,8.081,148.611
C02768=1172.033,311.511,-72.509,-176.700,8.078,148.611
C02769=1172.037,311.262,-72.478,-176.702,8.075,148.611
C02770=1172.041,311.015,-72.447,-176.705,8.072,148.611
C02771=1172.045,310.766,-72.415,-176.707,8.068,148.611
C02772=1172.050,310.518,-72.385,-176.710,8.065,148.611
C02773=1172.055,310.270,-72.354,-176.712,8.062,148.611
C02774=1172.058,310.023,-72.323,-176.715,8.059,148.611
C02775=1172.062,309.775,-72.292,-176.717,8.056,148.611
C02776=1172.067,309.527,-72.261,-176.720,8.053,148.611
C02777=1172.071,309.278,-72.230,-176.723,8.050,148.611
C02778=1172.075,309.030,-72.199,-176.725,8.047,148.610
C02779=1172.080,308.782,-72.169,-176.728,8.044,148.611
C02780=1172.083,308.534,-72.137,-176.730,8.041,148.611
C02781=1172.088,308.286,-72.107,-176.733,8.037,148.610
C02782=1172.092,308.038,-72.075,-176.735,8.034,148.610
C02783=1172.096,307.790,-72.045,-176.738,8.031,148.610
C02784=1172.100,307.542,-72.014,-176.740,8.028,148.610
C02785=1172.105,307.294,-71.984,-176.743,8.025,148.610
C02786=1172.109,307.045,-71.953,-176.745,8.022,148.610
C02787=1172.113,306.798,-71.922,-176.748,8.019,148.610
C02788=1172.117,306.550,-71.892,-176.751,8.016,148.610
C02789=1172.121,306.301,-71.860,-176.753,8.013,148.610
C02790=1172.126,306.053,-71.830,-176.756,8.010,148.610
C02791=1172.131,305.805,-71.799,-176.758,8.006,148.610
C02792=1172.134,305.557,-71.768,-176.760,8.004,148.610
C02793=1172.138,305.309,-71.738,-176.763,8.001,148.610
C02794=1172.143,305.061,-71.707,-176.765,7.998,148.610
C02795=1172.147,304.813,-71.677,-176.768,7.995,148.610
C02796=1172.151,304.565,-71.646,-176.771,7.992,148.610
C02797=1172.156,304.317,-71.615,-176.773,7.989,148.609
C02798=1172.159,304.069,-71.585,-176.776,7.986,148.609
C02799=1172.164,303.821,-71.554,-176.778,7.983,148.610
C02800=1172.168,303.572,-71.523,-176.781,7.979,148.609
C02801=1172.172,303.324,-71.493,-176.783,7.976,148.609
C02802=1172.177,303.076,-71.463,-176.786,7.973,148.609
C02803=1172.181,302.829,-71.432,-176.788,7.970,148.609
C02804=1172.185,302.581,-71.402,-176.791,7.967,148.609
C02805=1172.190,302.331,-71.371,-176.794,7.964,148.609
C02806=1172.193,302.084,-71.341,-176.796,7.961,148.609
C02807=1172.198,301.836,-71.310,-176.799,7.958,148.609
C02808=1172.202,301.588,-71.280,-176.802,7.955,148.609
C02809=1172.207,301.340,-71.249,-176.804,7.952,148.609
C02810=1172.210,301.091,-71.220,-176.807,7.949,148.609
C02811=1172.215,300.843,-71.189,-176.809,7.946,148.609
C02812=1172.219,300.596,-71.159,-176.812,7.942,148.609
C02813=1172.224,300.347,-71.129,-176.814,7.939,148.609
C02814=1172.227,300.099,-71.098,-176.817,7.936,148.609
C02815=1172.231,299.851,-71.067,-176.819,7.933,148.609
C02816=1172.236,299.602,-71.038,-176.822,7.930,148.609
C02817=1172.240,299.355,-71.007,-176.825,7.927,148.609
C02818=1172.244,299.107,-70.977,-176.828,7.924,148.609
C02819=1172.249,298.858,-70.947,-176.830,7.921,148.609
C02820=1172.253,298.611,-70.917,-176.832,7.919,148.609
C02821=1172.258,298.362,-70.887,-176.835,7.916,148.609
C02822=1172.261,298.114,-70.856,-176.837,7.912,148.608
C02823=1172.266,297.866,-70.825,-176.840,7.909,148.608
C02824=1172.270,297.617,-70.796,-176.843,7.906,148.608
C02825=1172.274,297.370,-70.766,-176.845,7.903,148.609
C02826=1172.279,297.121,-70.736,-176.848,7.900,148.608
C02827=1172.283,296.874,-70.705,-176.850,7.897,148.608
C02828=1172.288,296.625,-70.675,-176.853,7.894,148.608
C02829=1172.291,296.377,-70.645,-176.856,7.891,148.608
C02830=1172.296,296.129,-70.616,-176.858,7.888,148.608
C02831=1172.300,295.881,-70.585,-176.861,7.885,148.608
C02832=1172.304,295.632,-70.555,-176.864,7.882,148.608
C02833=1172.308,295.384,-70.526,-176.866,7.879,148.608
C02834=1172.313,295.136,-70.495,-176.869,7.876,148.608
C02835=1172.317,294.888,-70.466,-176.871,7.873,148.608
C02836=1172.321,294.640,-70.435,-176.874,7.870,148.608
C02837=1172.326,294.391,-70.405,-176.876,7.868,148.608
C02838=1172.330,294.143,-70.376,-176.879,7.864,148.608
C02839=1172.334,293.896,-70.346,-176.881,7.861,148.608
C02840=1172.338,293.647,-70.316,-176.884,7.858,148.608
C02841=1172.343,293.399,-70.286,-176.887,7.855,148.608
C02842=1172.347,293.151,-70.256,-176.889,7.852,148.608
C02843=1172.351,292.903,-70.227,-176.892,7.849,148.608
C02844=1172.355,292.655,-70.197,-176.895,7.846,148.608
C02845=1172.360,292.407,-70.166,-176.897,7.843,148.608
C02846=1172.364,292.158,-70.137,-176.900,7.840,148.608
C02847=1172.368,291.910,-70.107,-176.902,7.837,148.608
C02848=1172.372,291.662,-70.078,-176.904,7.835,148.608
C02849=1172.376,291.414,-70.049,-176.907,7.832,148.608
C02850=1172.381,291.166,-70.018,-176.910,7.829,148.608
C02851=1172.385,290.917,-69.988,-176.912,7.825,148.608
C02852=1172.389,290.669,-69.959,-176.915,7.822,148.608
C02853=1172.393,290.421,-69.929,-176.918,7.819,148.608
C02854=1172.398,290.172,-69.900,-176.920,7.816,148.608
C02855=1172.403,289.924,-69.870,-176.923,7.813,148.608
C02856=1172.406,289.676,-69.840,-176.925,7.810,148.608
C02857=1172.411,289.428,-69.810,-176.928,7.807,148.608
C02858=1172.415,289.180,-69.781,-176.931,7.804,148.608
C02859=1172.419,288.931,-69.751,-176.933,7.802,148.608
C02860=1172.423,288.683,-69.722,-176.936,7.799,148.608
C02861=1172.428,288.408,-69.689,-176.939,7.795,148.608
C02862=1172.433,288.134,-69.656,-176.941,7.792,148.608
C02863=1172.438,287.859,-69.624,-176.944,7.789,148.608
C02864=1172.442,287.584,-69.591,-176.947,7.785,148.608
C02865=1172.446,287.336,-69.562,-176.950,7.783,148.608
C02866=1172.451,287.087,-69.532,-176.952,7.780,148.608
C02867=1172.455,286.840,-69.503,-176.955,7.777,148.608
C02868=1172.459,286.592,-69.474,-176.958,7.774,148.608
C02869=1172.464,286.343,-69.444,-176.960,7.771,148.608
C02870=1172.468,286.095,-69.415,-176.963,7.768,148.608
C02871=1172.472,285.846,-69.386,-176.966,7.765,148.608
C02872=1172.477,285.598,-69.357,-176.968,7.762,148.608
C02873=1172.481,285.350,-69.327,-176.971,7.760,148.608
C02874=1172.485,285.101,-69.298,-176.973,7.757,148.608
C02875=1172.490,284.854,-69.269,-176.976,7.754,148.608
C02876=1172.494,284.605,-69.239,-176.978,7.751,148.608
C02877=1172.498,284.357,-69.210,-176.981,7.748,148.608
C02878=1172.502,284.109,-69.180,-176.984,7.745,148.608
C02879=1172.507,283.860,-69.151,-176.987,7.742,148.608
C02880=1172.511,283.612,-69.122,-176.989,7.739,148.608
C02881=1172.516,283.364,-69.093,-176.991,7.736,148.608
C02882=1172.520,283.116,-69.063,-176.994,7.733,148.608
C02883=1172.524,282.867,-69.035,-176.996,7.730,148.608
C02884=1172.528,282.619,-69.005,-176.999,7.727,148.608
C02885=1172.533,282.371,-68.976,-177.002,7.724,148.608
C02886=1172.537,282.123,-68.947,-177.005,7.721,148.608
C02887=1172.541,281.874,-68.919,-177.007,7.718,148.608
C02888=1172.545,281.626,-68.889,-177.010,7.716,148.608
C02889=1172.550,281.378,-68.860,-177.012,7.713,148.608
C02890=1172.554,281.129,-68.831,-177.015,7.710,148.608
C02891=1172.559,280.881,-68.802,-177.018,7.707,148.608
C02892=1172.563,280.633,-68.772,-177.020,7.704,148.608
C02893=1172.568,280.384,-68.744,-177.023,7.701,148.608
C02894=1172.571,280.136,-68.715,-177.026,7.698,148.608
C02895=1172.576,279.889,-68.686,-177.028,7.696,148.608
C02896=1172.580,279.640,-68.657,-177.030,7.693,148.608
C02897=1172.584,279.392,-68.627,-177.033,7.690,148.608
C02898=1172.588,279.143,-68.599,-177.036,7.687,148.609
C02899=1172.593,278.895,-68.570,-177.039,7.684,148.609
C02900=1172.597,278.647,-68.542,-177.041,7.681,148.609
C02901=1172.602,278.398,-68.512,-177.044,7.679,148.609
C02902=1172.606,278.149,-68.483,-177.046,7.676,148.609
C02903=1172.610,277.902,-68.455,-177.049,7.673,148.609
C02904=1172.615,277.653,-68.426,-177.051,7.670,148.609
C02905=1172.619,277.405,-68.397,-177.054,7.667,148.609
C02906=1172.623,277.157,-68.369,-177.057,7.664,148.609
C02907=1172.627,276.909,-68.339,-177.059,7.661,148.609
C02908=1172.632,276.660,-68.311,-177.062,7.659,148.609
C02909=1172.636,276.413,-68.282,-177.065,7.656,148.609
C02910=1172.640,276.164,-68.253,-177.067,7.653,148.609
C02911=1172.645,275.915,-68.225,-177.070,7.650,148.609
C02912=1172.650,275.667,-68.196,-177.073,7.647,148.609
C02913=1172.653,275.419,-68.167,-177.075,7.644,148.609
C02914=1172.658,275.171,-68.138,-177.078,7.641,148.609
C02915=1172.662,274.923,-68.110,-177.080,7.639,148.609
C02916=1172.666,274.674,-68.082,-177.083,7.636,148.609
C02917=1172.671,274.425,-68.052,-177.086,7.633,148.609
C02918=1172.675,274.178,-68.024,-177.088,7.630,148.609
C02919=1172.679,273.929,-67.996,-177.091,7.627,148.609
C02920=1172.684,273.680,-67.967,-177.094,7.624,148.609
C02921=1172.688,273.433,-67.938,-177.096,7.622,148.609
C02922=1172.692,273.184,-67.910,-177.099,7.618,148.609
C02923=1172.697,272.936,-67.882,-177.101,7.615,148.609
C02924=1172.701,272.687,-67.853,-177.103,7.613,148.609
C02925=1172.705,272.439,-67.824,-177.106,7.610,148.609
C02926=1172.710,272.191,-67.796,-177.109,7.607,148.610
C02927=1172.714,271.942,-67.768,-177.112,7.604,148.610
C02928=1172.719,271.694,-67.739,-177.114,7.602,148.610
C02929=1172.723,271.445,-67.711,-177.117,7.599,148.610
C02930=1172.727,271.197,-67.682,-177.119,7.596,148.610
C02931=1172.732,270.949,-67.653,-177.122,7.593,148.610
C02932=1172.735,270.700,-67.625,-177.125,7.590,148.610
C02933=1172.741,270.452,-67.597,-177.127,7.588,148.610
C02934=1172.744,270.204,-67.569,-177.130,7.585,148.610
C02935=1172.749,269.955,-67.540,-177.133,7.582,148.610
C02936=1172.753,269.707,-67.512,-177.135,7.579,148.610
C02937=1172.757,269.459,-67.484,-177.138,7.576,148.610
C02938=1172.762,269.210,-67.456,-177.140,7.574,148.610
C02939=1172.766,268.962,-67.428,-177.143,7.571,148.610
C02940=1172.771,268.713,-67.399,-177.146,7.568,148.610
C02941=1172.775,268.465,-67.371,-177.148,7.565,148.610
C02942=1172.780,268.217,-67.343,-177.151,7.563,148.610
C02943=1172.783,267.968,-67.314,-177.154,7.560,148.611
C02944=1172.788,267.720,-67.287,-177.157,7.557,148.611
C02945=1172.792,267.471,-67.258,-177.159,7.554,148.611
C02946=1172.797,267.223,-67.230,-177.162,7.551,148.611
C02947=1172.802,266.975,-67.202,-177.164,7.549,148.611
C02948=1172.805,266.727,-67.174,-177.167,7.546,148.611
C02949=1172.810,266.479,-67.146,-177.170,7.543,148.611
C02950=1172.814,266.230,-67.117,-177.172,7.540,148.611
C02951=1172.819,265.982,-67.089,-177.175,7.538,148.611
C02952=1172.822,265.733,-67.061,-177.177,7.535,148.611
C02953=1172.828,265.485,-67.034,-177.180,7.532,148.611
C02954=1172.831,265.236,-67.005,-177.183,7.529,148.611
C02955=1172.836,264.988,-66.978,-177.185,7.527,148.611
C02956=1172.840,264.739,-66.949,-177.188,7.524,148.611
C02957=1172.845,264.491,-66.921,-177.191,7.521,148.612
C02958=1172.849,264.243,-66.894,-177.193,7.518,148.612
C02959=1172.853,263.994,-66.866,-177.195,7.516,148.612
C02960=1172.858,263.746,-66.838,-177.198,7.513,148.612
C02961=1172.862,263.498,-66.809,-177.201,7.510,148.612
C02962=1172.867,263.249,-66.782,-177.204,7.507,148.612
C02963=1172.872,263.001,-66.754,-177.206,7.505,148.612
C02964=1172.875,262.752,-66.726,-177.209,7.502,148.612
C02965=1172.880,262.479,-66.695,-177.212,7.499,148.612
C02966=1172.885,262.206,-66.665,-177.215,7.496,148.612
C02967=1172.890,261.933,-66.634,-177.217,7.493,148.612
C02968=1172.895,261.660,-66.604,-177.221,7.490,148.612
C02969=1172.899,261.412,-66.576,-177.223,7.488,148.613
C02970=1172.904,261.163,-66.549,-177.226,7.485,148.613
C02971=1172.907,260.915,-66.521,-177.229,7.482,148.613
C02972=1172.912,260.667,-66.493,-177.231,7.480,148.613
C02973=1172.916,260.418,-66.466,-177.234,7.477,148.613
C02974=1172.921,260.169,-66.437,-177.236,7.474,148.613
C02975=1172.926,259.921,-66.410,-177.239,7.471,148.613
C02976=1172.930,259.673,-66.382,-177.241,7.469,148.613
C02977=1172.934,259.424,-66.355,-177.244,7.466,148.613
C02978=1172.938,259.176,-66.327,-177.247,7.463,148.613
C02979=1172.943,258.928,-66.300,-177.250,7.460,148.613
C02980=1172.947,258.679,-66.272,-177.252,7.458,148.614
C02981=1172.951,258.430,-66.245,-177.255,7.455,148.614
C02982=1172.956,258.183,-66.217,-177.258,7.452,148.614
C02983=1172.960,257.933,-66.189,-177.260,7.450,148.614
C02984=1172.964,257.686,-66.162,-177.263,7.447,148.614
C02985=1172.970,257.437,-66.134,-177.266,7.444,148.614
C02986=1172.973,257.188,-66.106,-177.268,7.442,148.614
C02987=1172.978,256.940,-66.079,-177.271,7.439,148.614
C02988=1172.983,256.691,-66.052,-177.274,7.436,148.614
C02989=1172.987,256.443,-66.024,-177.276,7.433,148.614
C02990=1172.991,256.194,-65.997,-177.278,7.431,148.614
C02991=1172.995,255.946,-65.969,-177.281,7.428,148.615
C02992=1173.000,255.698,-65.942,-177.284,7.426,148.615
C02993=1173.005,255.449,-65.915,-177.287,7.423,148.615
C02994=1173.008,255.201,-65.886,-177.289,7.420,148.615
C02995=1173.013,254.952,-65.859,-177.292,7.417,148.615
C02996=1173.018,254.704,-65.832,-177.294,7.415,148.615
C02997=1173.022,254.455,-65.805,-177.297,7.412,148.615
C02998=1173.025,254.207,-65.778,-177.300,7.410,148.615
C02999=1173.030,253.958,-65.751,-177.302,7.408,148.616
C03000=1173.035,253.710,-65.724,-177.305,7.405,148.616
C03001=1173.039,253.461,-65.697,-177.308,7.402,148.616
C03002=1173.044,253.214,-65.669,-177.311,7.399,148.616
C03003=1173.048,252.964,-65.641,-177.313,7.397,148.616
C03004=1173.052,252.716,-65.614,-177.316,7.394,148.616
C03005=1173.057,252.467,-65.587,-177.319,7.391,148.616
C03006=1173.062,252.219,-65.560,-177.321,7.389,148.616
C03007=1173.066,251.971,-65.532,-177.324,7.386,148.616
C03008=1173.069,251.722,-65.506,-177.326,7.383,148.616
C03009=1173.074,251.474,-65.479,-177.329,7.381,148.617
C03010=1173.079,251.225,-65.451,-177.332,7.378,148.617
C03011=1173.083,250.977,-65.424,-177.335,7.375,148.617
C03012=1173.088,250.728,-65.397,-177.337,7.373,148.617
C03013=1173.093,250.480,-65.370,-177.340,7.370,148.617
C03014=1173.097,250.231,-65.344,-177.343,7.367,148.617
C03015=1173.101,249.982,-65.316,-177.345,7.365,148.617
C03016=1173.105,249.734,-65.289,-177.348,7.362,148.617
C03017=1173.110,249.485,-65.262,-177.350,7.360,148.618
C03018=1173.115,249.237,-65.235,-177.353,7.358,148.618
C03019=1173.119,248.989,-65.209,-177.356,7.355,148.618
C03020=1173.123,248.740,-65.182,-177.358,7.352,148.618
C03021=1173.128,248.492,-65.155,-177.361,7.349,148.618
C03022=1173.133,248.243,-65.128,-177.364,7.347,148.618
C03023=1173.136,247.995,-65.101,-177.366,7.345,148.618
C03024=1173.141,247.746,-65.074,-177.369,7.342,148.618
C03025=1173.145,247.497,-65.047,-177.372,7.339,148.619
C03026=1173.150,247.249,-65.020,-177.374,7.337,148.619
C03027=1173.154,247.000,-64.993,-177.377,7.334,148.619
C03028=1173.158,246.752,-64.966,-177.380,7.331,148.619
C03029=1173.163,246.503,-64.939,-177.382,7.329,148.619
C03030=1173.167,246.255,-64.912,-177.385,7.326,148.619
C03031=1173.172,246.007,-64.885,-177.387,7.324,148.619
C03032=1173.177,245.758,-64.859,-177.390,7.321,148.620
C03033=1173.181,245.510,-64.833,-177.393,7.318,148.620
C03034=1173.185,245.261,-64.806,-177.396,7.316,148.620
C03035=1173.190,245.013,-64.778,-177.398,7.313,148.620
C03036=1173.194,244.764,-64.752,-177.400,7.311,148.620
C03037=1173.199,244.515,-64.726,-177.404,7.309,148.620
C03038=1173.203,244.267,-64.699,-177.406,7.306,148.620
C03039=1173.207,244.019,-64.672,-177.409,7.304,148.621
C03040=1173.212,243.770,-64.645,-177.411,7.301,148.621
C03041=1173.216,243.521,-64.619,-177.415,7.298,148.621
C03042=1173.221,243.273,-64.592,-177.417,7.296,148.621
C03043=1173.225,243.025,-64.566,-177.420,7.293,148.621
C03044=1173.230,242.775,-64.539,-177.422,7.291,148.621
C03045=1173.234,242.527,-64.513,-177.425,7.288,148.621
C03046=1173.238,242.279,-64.486,-177.428,7.285,148.622
C03047=1173.243,242.030,-64.460,-177.430,7.283,148.622
C03048=1173.247,241.781,-64.433,-177.433,7.280,148.622
C03049=1173.252,241.533,-64.406,-177.435,7.278,148.622
C03050=1173.256,241.284,-64.380,-177.438,7.275,148.622
C03051=1173.261,241.036,-64.353,-177.441,7.273,148.622
C03052=1173.265,240.787,-64.327,-177.443,7.270,148.622
C03053=1173.270,240.538,-64.300,-177.446,7.268,148.623
C03054=1173.273,240.290,-64.274,-177.449,7.266,148.623
C03055=1173.278,240.041,-64.248,-177.452,7.263,148.623
C03056=1173.282,239.793,-64.221,-177.454,7.261,148.623
C03057=1173.287,239.544,-64.195,-177.457,7.258,148.623
C03058=1173.291,239.296,-64.168,-177.460,7.255,148.623
C03059=1173.295,239.047,-64.143,-177.462,7.253,148.623
C03060=1173.301,238.799,-64.116,-177.465,7.250,148.624
C03061=1173.305,238.550,-64.090,-177.467,7.248,148.624
C03062=1173.310,238.302,-64.063,-177.470,7.245,148.624
C03063=1173.314,238.053,-64.037,-177.473,7.243,148.624
C03064=1173.319,237.804,-64.010,-177.475,7.240,148.624
C03065=1173.323,237.556,-63.985,-177.479,7.238,148.625
C03066=1173.327,237.307,-63.959,-177.481,7.236,148.625
C03067=1173.332,237.058,-63.932,-177.484,7.233,148.625
C03068=1173.336,236.809,-63.906,-177.486,7.231,148.625
C03069=1173.341,236.539,-63.878,-177.489,7.228,148.625
C03070=1173.346,236.267,-63.849,-177.492,7.225,148.626
C03071=1173.351,235.995,-63.820,-177.495,7.222,148.626
C03072=1173.355,235.723,-63.792,-177.498,7.220,148.626
C03073=1173.360,235.475,-63.765,-177.500,7.218,148.626
C03074=1173.364,235.226,-63.739,-177.503,7.215,148.626
C03075=1173.368,234.977,-63.714,-177.506,7.213,148.626
C03076=1173.374,234.730,-63.687,-177.509,7.210,148.626
C03077=1173.378,234.481,-63.661,-177.512,7.207,148.627
C03078=1173.382,234.232,-63.635,-177.514,7.205,148.627
C03079=1173.387,233.983,-63.609,-177.517,7.202,148.627
C03080=1173.391,233.735,-63.583,-177.519,7.200,148.627
C03081=1173.396,233.487,-63.557,-177.522,7.197,148.627
C03082=1173.400,233.238,-63.531,-177.525,7.196,148.628
C03083=1173.405,232.989,-63.505,-177.528,7.193,148.628
C03084=1173.409,232.740,-63.479,-177.530,7.190,148.628
C03085=1173.413,232.492,-63.453,-177.533,7.188,148.628
C03086=1173.418,232.244,-63.427,-177.535,7.186,148.628
C03087=1173.422,231.995,-63.402,-177.538,7.183,148.629
C03088=1173.427,231.746,-63.375,-177.541,7.181,148.629
C03089=1173.431,231.497,-63.350,-177.543,7.178,148.629
C03090=1173.436,231.249,-63.324,-177.546,7.176,148.629
C03091=1173.440,231.000,-63.298,-177.549,7.173,148.629
C03092=1173.445,230.751,-63.273,-177.552,7.171,148.629
C03093=1173.450,230.502,-63.246,-177.554,7.168,148.630
C03094=1173.454,230.255,-63.220,-177.557,7.166,148.630
C03095=1173.458,230.006,-63.195,-177.560,7.164,148.630
C03096=1173.463,229.757,-63.169,-177.562,7.161,148.630
C03097=1173.467,229.508,-63.143,-177.565,7.159,148.630
C03098=1173.472,229.260,-63.118,-177.568,7.156,148.630
C03099=1173.476,229.011,-63.092,-177.570,7.154,148.631
C03100=1173.480,228.762,-63.066,-177.573,7.151,148.631
C03101=1173.486,228.514,-63.040,-177.576,7.149,148.631
C03102=1173.490,228.265,-63.014,-177.579,7.147,148.631
C03103=1173.494,228.016,-62.989,-177.581,7.145,148.632
C03104=1173.499,227.768,-62.963,-177.584,7.142,148.632
C03105=1173.503,227.519,-62.938,-177.587,7.140,148.632
C03106=1173.508,227.270,-62.912,-177.589,7.137,148.632
C03107=1173.512,227.021,-62.887,-177.592,7.135,148.632
C03108=1173.517,226.773,-62.861,-177.595,7.132,148.632
C03109=1173.521,226.524,-62.836,-177.597,7.130,148.633
C03110=1173.526,226.276,-62.810,-177.600,7.128,148.633
C03111=1173.530,226.027,-62.784,-177.602,7.125,148.633
C03112=1173.534,225.779,-62.759,-177.605,7.124,148.633
C03113=1173.539,225.530,-62.734,-177.608,7.121,148.633
C03114=1173.544,225.281,-62.708,-177.610,7.119,148.634
C03115=1173.548,225.032,-62.683,-177.613,7.116,148.634
C03116=1173.553,224.784,-62.657,-177.616,7.114,148.634
C03117=1173.557,224.535,-62.631,-177.619,7.111,148.634
C03118=1173.561,224.286,-62.606,-177.621,7.109,148.635
C03119=1173.566,224.038,-62.581,-177.624,7.106,148.635
C03120=1173.570,223.789,-62.555,-177.627,7.105,148.635
C03121=1173.575,223.541,-62.530,-177.629,7.102,148.635
C03122=1173.580,223.292,-62.505,-177.632,7.100,148.635
C03123=1173.584,223.043,-62.479,-177.635,7.097,148.635
C03124=1173.588,222.795,-62.454,-177.638,7.095,148.636
C03125=1173.593,222.545,-62.429,-177.640,7.093,148.636
C03126=1173.598,222.297,-62.404,-177.643,7.090,148.636
C03127=1173.602,222.049,-62.378,-177.645,7.088,148.636
C03128=1173.607,221.800,-62.353,-177.648,7.086,148.637
C03129=1173.611,221.551,-62.328,-177.651,7.083,148.637
C03130=1173.615,221.302,-62.302,-177.654,7.081,148.637
C03131=1173.620,221.054,-62.277,-177.656,7.079,148.637
C03132=1173.624,220.805,-62.252,-177.659,7.076,148.637
C03133=1173.629,220.556,-62.227,-177.661,7.074,148.638
C03134=1173.633,220.308,-62.202,-177.665,7.071,148.638
C03135=1173.638,220.059,-62.176,-177.667,7.069,148.638
C03136=1173.643,219.810,-62.151,-177.670,7.067,148.638
C03137=1173.647,219.562,-62.126,-177.673,7.065,148.639
C03138=1173.651,219.313,-62.101,-177.675,7.063,148.639
C03139=1173.656,219.065,-62.076,-177.678,7.060,148.639
C03140=1173.661,218.815,-62.051,-177.680,7.058,148.639
C03141=1173.665,218.567,-62.026,-177.684,7.055,148.639
C03142=1173.669,218.318,-62.001,-177.686,7.053,148.640
C03143=1173.674,218.070,-61.976,-177.688,7.051,148.640
C03144=1173.679,217.820,-61.951,-177.691,7.048,148.640
C03145=1173.683,217.572,-61.925,-177.694,7.047,148.640
C03146=1173.687,217.323,-61.901,-177.697,7.044,148.641
C03147=1173.692,217.075,-61.876,-177.699,7.042,148.641
C03148=1173.697,216.826,-61.851,-177.702,7.040,148.641
C03149=1173.701,216.577,-61.826,-177.705,7.037,148.641
C03150=1173.705,216.329,-61.801,-177.707,7.035,148.642
C03151=1173.710,216.080,-61.776,-177.710,7.032,148.642
C03152=1173.715,215.830,-61.751,-177.713,7.031,148.642
C03153=1173.719,215.583,-61.726,-177.715,7.028,148.642
C03154=1173.724,215.334,-61.702,-177.718,7.026,148.642
C03155=1173.729,215.084,-61.677,-177.721,7.024,148.643
C03156=1173.733,214.837,-61.652,-177.724,7.021,148.643
C03157=1173.737,214.587,-61.627,-177.726,7.019,148.643
C03158=1173.742,214.339,-61.603,-177.728,7.017,148.643
C03159=1173.746,214.089,-61.578,-177.732,7.015,148.644
C03160=1173.751,213.841,-61.552,-177.734,7.013,148.644
C03161=1173.755,213.593,-61.528,-177.737,7.010,148.644
C03162=1173.760,213.343,-61.503,-177.740,7.008,148.644
C03163=1173.765,213.095,-61.478,-177.742,7.006,148.644
C03164=1173.769,212.846,-61.453,-177.745,7.003,148.645
C03165=1173.774,212.597,-61.429,-177.747,7.001,148.645
C03166=1173.778,212.349,-61.405,-177.751,6.999,148.645
C03167=1173.783,212.100,-61.379,-177.753,6.997,148.646
C03168=1173.787,211.851,-61.355,-177.756,6.995,148.646
C03169=1173.792,211.603,-61.331,-177.759,6.992,148.646
C03170=1173.796,211.354,-61.306,-177.761,6.990,148.646
C03171=1173.801,211.105,-61.281,-177.764,6.988,148.646
C03172=1173.806,210.857,-61.256,-177.767,6.985,148.647
C03173=1173.810,210.586,-61.230,-177.770,6.983,148.647
C03174=1173.815,210.316,-61.203,-177.772,6.981,148.647
C03175=1173.820,210.045,-61.177,-177.776,6.978,148.647
C03176=1173.825,209.774,-61.150,-177.778,6.976,148.648
C03177=1173.830,209.525,-61.125,-177.781,6.973,148.648
C03178=1173.834,209.277,-61.101,-177.784,6.972,148.648
C03179=1173.839,209.028,-61.076,-177.787,6.969,148.649
C03180=1173.843,208.779,-61.052,-177.789,6.967,148.649
C03181=1173.848,208.530,-61.027,-177.792,6.965,148.649
C03182=1173.852,208.281,-61.003,-177.795,6.962,148.649
C03183=1173.857,208.033,-60.978,-177.797,6.960,148.649
C03184=1173.862,207.784,-60.954,-177.800,6.959,148.650
C03185=1173.866,207.536,-60.930,-177.803,6.956,148.650
C03186=1173.871,207.286,-60.905,-177.805,6.954,148.650
C03187=1173.875,207.038,-60.881,-177.808,6.952,148.651
C03188=1173.880,206.789,-60.856,-177.811,6.949,148.651
C03189=1173.885,206.541,-60.832,-177.813,6.947,148.651
C03190=1173.888,206.292,-60.808,-177.816,6.946,148.651
C03191=1173.894,206.043,-60.783,-177.819,6.943,148.651
C03192=1173.898,205.795,-60.759,-177.821,6.941,148.652
C03193=1173.902,205.546,-60.735,-177.824,6.939,148.652
C03194=1173.907,205.296,-60.711,-177.827,6.936,148.652
C03195=1173.912,205.048,-60.687,-177.830,6.934,148.653
C03196=1173.917,204.799,-60.662,-177.832,6.932,148.653
C03197=1173.921,204.551,-60.638,-177.835,6.930,148.653
C03198=1173.925,204.301,-60.613,-177.838,6.928,148.653
C03199=1173.930,204.052,-60.590,-177.840,6.926,148.654
C03200=1173.935,203.804,-60.565,-177.843,6.923,148.654
C03201=1173.939,203.555,-60.541,-177.846,6.921,148.654
C03202=1173.943,203.307,-60.517,-177.848,6.919,148.655
C03203=1173.948,203.057,-60.493,-177.851,6.916,148.655
C03204=1173.953,202.808,-60.469,-177.854,6.915,148.655
C03205=1173.957,202.560,-60.445,-177.856,6.913,148.655
C03206=1173.961,202.312,-60.421,-177.859,6.910,148.655
C03207=1173.967,202.062,-60.397,-177.862,6.908,148.656
C03208=1173.971,201.814,-60.373,-177.865,6.906,148.656
C03209=1173.975,201.565,-60.348,-177.867,6.904,148.656
C03210=1173.980,201.316,-60.325,-177.870,6.902,148.657
C03211=1173.984,201.067,-60.301,-177.873,6.900,148.657
C03212=1173.989,200.819,-60.276,-177.875,6.898,148.657
C03213=1173.994,200.570,-60.253,-177.878,6.895,148.657
C03214=1173.998,200.321,-60.229,-177.881,6.893,148.658
C03215=1174.003,200.071,-60.205,-177.883,6.891,148.658
C03216=1174.007,199.823,-60.181,-177.886,6.889,148.658
C03217=1174.012,199.574,-60.156,-177.889,6.887,148.658
C03218=1174.017,199.325,-60.133,-177.892,6.885,148.659
C03219=1174.021,199.077,-60.109,-177.894,6.883,148.659
C03220=1174.026,198.828,-60.086,-177.897,6.880,148.659
C03221=1174.030,198.579,-60.061,-177.900,6.879,148.660
C03222=1174.035,198.330,-60.038,-177.902,6.876,148.660
C03223=1174.039,198.082,-60.014,-177.905,6.874,148.660
C03224=1174.044,197.833,-59.991,-177.908,6.872,148.660
C03225=1174.049,197.583,-59.966,-177.910,6.870,148.661
C03226=1174.053,197.334,-59.942,-177.913,6.868,148.661
C03227=1174.058,197.086,-59.918,-177.916,6.866,148.661
C03228=1174.062,196.837,-59.895,-177.919,6.864,148.662
C03229=1174.067,196.589,-59.871,-177.921,6.862,148.662
C03230=1174.071,196.340,-59.847,-177.923,6.860,148.662
C03231=1174.076,196.091,-59.824,-177.927,6.857,148.662
C03232=1174.081,195.842,-59.800,-177.929,6.855,148.663
C03233=1174.085,195.593,-59.777,-177.932,6.853,148.663
C03234=1174.090,195.345,-59.753,-177.935,6.851,148.663
C03235=1174.094,195.096,-59.729,-177.937,6.849,148.664
C03236=1174.099,194.847,-59.706,-177.940,6.847,148.664
C03237=1174.103,194.598,-59.682,-177.942,6.845,148.664
C03238=1174.108,194.349,-59.658,-177.946,6.842,148.664
C03239=1174.113,194.100,-59.635,-177.948,6.841,148.665
C03240=1174.117,193.852,-59.611,-177.951,6.839,148.665
C03241=1174.122,193.603,-59.588,-177.953,6.837,148.665
C03242=1174.127,193.354,-59.564,-177.956,6.834,148.665
C03243=1174.131,193.105,-59.541,-177.959,6.832,148.666
C03244=1174.136,192.856,-59.517,-177.962,6.831,148.666
C03245=1174.140,192.607,-59.493,-177.964,6.829,148.666
C03246=1174.145,192.358,-59.470,-177.967,6.826,148.667
C03247=1174.150,192.109,-59.447,-177.970,6.824,148.667
C03248=1174.154,191.861,-59.423,-177.973,6.822,148.667
C03249=1174.159,191.612,-59.399,-177.975,6.820,148.668
C03250=1174.164,191.363,-59.376,-177.977,6.818,148.668
C03251=1174.168,191.114,-59.353,-177.981,6.816,148.668
C03252=1174.172,190.865,-59.330,-177.983,6.814,148.669
C03253=1174.177,190.616,-59.306,-177.985,6.812,148.669
C03254=1174.181,190.367,-59.282,-177.988,6.810,148.669
C03255=1174.186,190.118,-59.259,-177.991,6.808,148.669
C03256=1174.191,189.869,-59.236,-177.994,6.806,148.670
C03257=1174.195,189.620,-59.212,-177.996,6.804,148.670
C03258=1174.201,189.372,-59.189,-177.999,6.802,148.670
C03259=1174.205,189.123,-59.167,-178.002,6.800,148.671
C03260=1174.209,188.874,-59.143,-178.005,6.798,148.671
C03261=1174.214,188.625,-59.120,-178.008,6.796,148.671
C03262=1174.219,188.376,-59.096,-178.010,6.794,148.671
C03263=1174.224,188.127,-59.073,-178.012,6.792,148.672
C03264=1174.228,187.878,-59.050,-178.016,6.789,148.672
C03265=1174.232,187.629,-59.027,-178.018,6.787,148.672
C03266=1174.237,187.380,-59.004,-178.021,6.786,148.673
C03267=1174.242,187.131,-58.980,-178.023,6.784,148.673
C03268=1174.247,186.883,-58.957,-178.026,6.782,148.673
C03269=1174.251,186.634,-58.934,-178.029,6.779,148.674
C03270=1174.256,186.385,-58.911,-178.032,6.777,148.674
C03271=1174.260,186.136,-58.888,-178.035,6.776,148.674
C03272=1174.265,185.887,-58.864,-178.037,6.774,148.674
C03273=1174.269,185.638,-58.842,-178.039,6.772,148.675
C03274=1174.274,185.389,-58.818,-178.043,6.769,148.675
C03275=1174.279,185.141,-58.795,-178.045,6.767,148.675
C03276=1174.284,184.892,-58.772,-178.048,6.766,148.676
C03277=1174.288,184.623,-58.747,-178.051,6.764,148.676
C03278=1174.294,184.353,-58.722,-178.054,6.761,148.677
C03279=1174.298,184.083,-58.698,-178.057,6.759,148.677
C03280=1174.303,183.814,-58.673,-178.060,6.757,148.677
C03281=1174.308,183.565,-58.650,-178.062,6.755,148.677
C03282=1174.312,183.316,-58.627,-178.065,6.753,148.678
C03283=1174.317,183.067,-58.604,-178.067,6.751,148.678
C03284=1174.322,182.819,-58.581,-178.070,6.749,148.678
C03285=1174.326,182.569,-58.558,-178.073,6.747,148.679
C03286=1174.331,182.320,-58.535,-178.076,6.745,148.679
C03287=1174.336,182.071,-58.512,-178.078,6.743,148.679
C03288=1174.340,181.822,-58.489,-178.081,6.741,148.680
C03289=1174.345,181.573,-58.467,-178.084,6.739,148.680
C03290=1174.349,181.325,-58.444,-178.086,6.738,148.680
C03291=1174.354,181.076,-58.421,-178.089,6.735,148.681
C03292=1174.359,180.826,-58.398,-178.092,6.733,148.681
C03293=1174.364,180.578,-58.376,-178.094,6.731,148.681
C03294=1174.368,180.329,-58.352,-178.097,6.729,148.682
C03295=1174.373,180.080,-58.330,-178.100,6.728,148.682
C03296=1174.377,179.831,-58.307,-178.102,6.726,148.682
C03297=1174.382,179.583,-58.284,-178.105,6.724,148.683
C03298=1174.387,179.333,-58.262,-178.108,6.721,148.683
C03299=1174.391,179.084,-58.239,-178.111,6.720,148.683
C03300=1174.395,178.835,-58.216,-178.113,6.718,148.683
C03301=1174.400,178.587,-58.194,-178.116,6.716,148.684
C03302=1174.405,178.338,-58.171,-178.119,6.714,148.684
C03303=1174.409,178.088,-58.149,-178.121,6.712,148.685
C03304=1174.415,177.840,-58.126,-178.124,6.711,148.685
C03305=1174.419,177.590,-58.103,-178.127,6.708,148.685
C03306=1174.424,177.341,-58.080,-178.130,6.706,148.686
C03307=1174.428,177.093,-58.058,-178.132,6.704,148.686
C03308=1174.433,176.844,-58.035,-178.135,6.702,148.686
C03309=1174.437,176.595,-58.012,-178.137,6.701,148.686
C03310=1174.443,176.346,-57.990,-178.140,6.699,148.687
C03311=1174.447,176.097,-57.967,-178.143,6.697,148.687
C03312=1174.451,175.848,-57.945,-178.145,6.695,148.688
C03313=1174.457,175.599,-57.923,-178.149,6.693,148.688
C03314=1174.460,175.350,-57.900,-178.151,6.691,148.688
C03315=1174.465,175.101,-57.878,-178.154,6.689,148.689
C03316=1174.470,174.853,-57.855,-178.156,6.687,148.689
C03317=1174.474,174.603,-57.833,-178.159,6.685,148.689
C03318=1174.479,174.354,-57.810,-178.162,6.683,148.689
C03319=1174.484,174.106,-57.788,-178.164,6.682,148.690
C03320=1174.489,173.856,-57.765,-178.167,6.680,148.690
C03321=1174.493,173.607,-57.743,-178.170,6.678,148.691
C03322=1174.498,173.359,-57.721,-178.173,6.676,148.691
C03323=1174.503,173.109,-57.698,-178.176,6.674,148.691
C03324=1174.507,172.861,-57.676,-178.178,6.672,148.692
C03325=1174.512,172.612,-57.654,-178.181,6.670,148.692
C03326=1174.517,172.362,-57.631,-178.183,6.668,148.692
C03327=1174.521,172.114,-57.609,-178.186,6.666,148.693
C03328=1174.525,171.865,-57.587,-178.189,6.665,148.693
C03329=1174.531,171.616,-57.565,-178.191,6.663,148.693
C03330=1174.535,171.367,-57.542,-178.194,6.661,148.694
C03331=1174.540,171.118,-57.520,-178.197,6.659,148.694
C03332=1174.544,170.869,-57.498,-178.200,6.657,148.694
C03333=1174.550,170.620,-57.476,-178.203,6.655,148.695
C03334=1174.554,170.371,-57.453,-178.205,6.653,148.695
C03335=1174.558,170.122,-57.431,-178.208,6.651,148.695
C03336=1174.563,169.873,-57.409,-178.211,6.650,148.696
C03337=1174.568,169.624,-57.387,-178.213,6.648,148.696
C03338=1174.573,169.375,-57.365,-178.215,6.646,148.696
C03339=1174.577,169.126,-57.343,-178.218,6.644,148.697
C03340=1174.582,168.878,-57.320,-178.221,6.642,148.697
C03341=1174.587,168.628,-57.298,-178.224,6.640,148.697
C03342=1174.591,168.379,-57.276,-178.226,6.639,148.698
C03343=1174.596,168.130,-57.254,-178.229,6.637,148.698
C03344=1174.601,167.881,-57.232,-178.232,6.635,148.699
C03345=1174.605,167.632,-57.210,-178.235,6.633,148.699
C03346=1174.610,167.383,-57.188,-178.238,6.631,148.699
C03347=1174.615,167.134,-57.166,-178.240,6.629,148.700
C03348=1174.620,166.885,-57.144,-178.243,6.627,148.700
C03349=1174.624,166.636,-57.122,-178.246,6.626,148.700
C03350=1174.628,166.388,-57.100,-178.248,6.624,148.701
C03351=1174.633,166.138,-57.078,-178.251,6.622,148.701
C03352=1174.638,165.890,-57.056,-178.254,6.620,148.701
C03353=1174.642,165.640,-57.034,-178.256,6.618,148.702
C03354=1174.647,165.392,-57.012,-178.259,6.617,148.702
C03355=1174.652,165.143,-56.990,-178.262,6.615,148.703
C03356=1174.657,164.894,-56.968,-178.264,6.613,148.703
C03357=1174.661,164.645,-56.946,-178.267,6.611,148.703
C03358=1174.666,164.395,-56.925,-178.269,6.609,148.703
C03359=1174.671,164.146,-56.903,-178.272,6.608,148.704
C03360=1174.675,163.897,-56.881,-178.275,6.606,148.704
C03361=1174.680,163.648,-56.860,-178.277,6.604,148.705
C03362=1174.684,163.399,-56.838,-178.280,6.602,148.705
C03363=1174.689,163.150,-56.816,-178.283,6.601,148.705
C03364=1174.694,162.902,-56.794,-178.285,6.599,148.706
C03365=1174.698,162.652,-56.772,-178.288,6.597,148.706
C03366=1174.703,162.404,-56.751,-178.291,6.595,148.706
C03367=1174.707,162.154,-56.729,-178.293,6.593,148.707
C03368=1174.713,161.905,-56.708,-178.296,6.592,148.707
C03369=1174.717,161.656,-56.686,-178.299,6.589,148.708
C03370=1174.722,161.407,-56.664,-178.302,6.587,148.708
C03371=1174.727,161.158,-56.642,-178.305,6.586,148.708
C03372=1174.731,160.910,-56.620,-178.307,6.584,148.709
C03373=1174.736,160.660,-56.599,-178.310,6.582,148.709
C03374=1174.741,160.411,-56.577,-178.313,6.580,148.709
C03375=1174.745,160.162,-56.555,-178.316,6.579,148.710
C03376=1174.750,159.913,-56.534,-178.318,6.577,148.710
C03377=1174.755,159.664,-56.513,-178.321,6.575,148.711
C03378=1174.759,159.415,-56.491,-178.324,6.573,148.711
C03379=1174.764,159.166,-56.469,-178.326,6.572,148.711
C03380=1174.769,158.917,-56.447,-178.329,6.570,148.712
C03381=1174.774,158.648,-56.425,-178.332,6.568,148.712
C03382=1174.779,158.379,-56.401,-178.334,6.566,148.712
C03383=1174.784,158.110,-56.378,-178.338,6.565,148.713
C03384=1174.789,157.841,-56.354,-178.341,6.562,148.713
C03385=1174.794,157.592,-56.334,-178.343,6.561,148.714
C03386=1174.798,157.343,-56.312,-178.346,6.559,148.714
C03387=1174.803,157.094,-56.290,-178.349,6.557,148.714
C03388=1174.808,156.845,-56.269,-178.352,6.555,148.715
C03389=1174.813,156.596,-56.248,-178.354,6.553,148.715
C03390=1174.818,156.346,-56.226,-178.357,6.552,148.716
C03391=1174.822,156.098,-56.205,-178.360,6.550,148.716
C03392=1174.827,155.849,-56.184,-178.362,6.549,148.716
C03393=1174.831,155.599,-56.162,-178.364,6.547,148.717
C03394=1174.836,155.351,-56.140,-178.367,6.546,148.717
C03395=1174.841,155.102,-56.120,-178.370,6.544,148.717
C03396=1174.846,154.853,-56.098,-178.372,6.542,148.718
C03397=1174.850,154.603,-56.077,-178.375,6.540,148.718
C03398=1174.855,154.355,-56.055,-178.378,6.538,148.719
C03399=1174.860,154.105,-56.034,-178.381,6.537,148.719
C03400=1174.865,153.857,-56.013,-178.383,6.535,148.719
C03401=1174.869,153.607,-55.992,-178.386,6.533,148.720
C03402=1174.873,153.358,-55.970,-178.389,6.531,148.720
C03403=1174.879,153.109,-55.949,-178.391,6.530,148.720
C03404=1174.884,152.861,-55.928,-178.394,6.528,148.721
C03405=1174.888,152.612,-55.907,-178.397,6.526,148.721
C03406=1174.893,152.362,-55.886,-178.400,6.525,148.722
C03407=1174.897,152.113,-55.864,-178.403,6.523,148.722
C03408=1174.903,151.864,-55.843,-178.405,6.521,148.723
C03409=1174.907,151.615,-55.822,-178.408,6.520,148.723
C03410=1174.912,151.366,-55.801,-178.411,6.518,148.723
C03411=1174.916,151.116,-55.780,-178.413,6.516,148.724
C03412=1174.921,150.868,-55.759,-178.416,6.514,148.724
C03413=1174.926,150.619,-55.738,-178.419,6.513,148.725
C03414=1174.931,150.369,-55.717,-178.421,6.511,148.725
C03415=1174.935,150.121,-55.696,-178.424,6.509,148.725
C03416=1174.940,149.872,-55.675,-178.427,6.507,148.726
C03417=1174.945,149.622,-55.654,-178.429,6.506,148.726
C03418=1174.949,149.373,-55.632,-178.432,6.505,148.726
C03419=1174.954,149.124,-55.611,-178.434,6.503,148.727
C03420=1174.959,148.875,-55.591,-178.437,6.501,148.727
C03421=1174.964,148.626,-55.570,-178.440,6.499,148.728
C03422=1174.969,148.377,-55.548,-178.443,6.498,148.728
C03423=1174.973,148.128,-55.528,-178.446,6.496,148.729
C03424=1174.978,147.879,-55.507,-178.448,6.494,148.729
C03425=1174.982,147.629,-55.486,-178.451,6.493,148.729
C03426=1174.987,147.381,-55.465,-178.454,6.491,148.730
C03427=1174.992,147.132,-55.444,-178.456,6.489,148.730
C03428=1174.997,146.883,-55.423,-178.459,6.487,148.730
C03429=1175.002,146.633,-55.402,-178.462,6.486,148.731
C03430=1175.006,146.384,-55.382,-178.464,6.485,148.731
C03431=1175.011,146.135,-55.361,-178.467,6.483,148.732
C03432=1175.015,145.887,-55.340,-178.469,6.481,148.732
C03433=1175.021,145.638,-55.319,-178.472,6.479,148.732
C03434=1175.025,145.389,-55.299,-178.475,6.478,148.733
C03435=1175.030,145.139,-55.278,-178.478,6.476,148.733
C03436=1175.034,144.890,-55.257,-178.480,6.475,148.734
C03437=1175.039,144.640,-55.236,-178.483,6.473,148.734
C03438=1175.044,144.392,-55.216,-178.486,6.471,148.735
C03439=1175.049,144.142,-55.195,-178.489,6.469,148.735
C03440=1175.053,143.893,-55.174,-178.491,6.468,148.735
C03441=1175.058,143.644,-55.153,-178.493,6.467,148.736
C03442=1175.063,143.395,-55.133,-178.496,6.465,148.736
C03443=1175.067,143.146,-55.113,-178.499,6.463,148.737
C03444=1175.073,142.897,-55.092,-178.502,6.462,148.737
C03445=1175.077,142.648,-55.071,-178.505,6.460,148.737
C03446=1175.082,142.399,-55.050,-178.507,6.458,148.738
C03447=1175.087,142.150,-55.030,-178.510,6.456,148.738
C03448=1175.092,141.900,-55.009,-178.513,6.455,148.739
C03449=1175.096,141.652,-54.989,-178.515,6.453,148.739
C03450=1175.101,141.403,-54.968,-178.518,6.452,148.739
C03451=1175.106,141.153,-54.947,-178.520,6.450,148.740
C03452=1175.110,140.904,-54.927,-178.523,6.449,148.740
C03453=1175.115,140.655,-54.906,-178.526,6.447,148.741
C03454=1175.120,140.406,-54.885,-178.529,6.445,148.741
C03455=1175.124,140.157,-54.865,-178.532,6.444,148.742
C03456=1175.129,139.908,-54.844,-178.534,6.442,148.742
C03457=1175.134,139.658,-54.824,-178.537,6.440,148.742
C03458=1175.139,139.409,-54.804,-178.539,6.439,148.743
C03459=1175.144,139.160,-54.783,-178.542,6.438,148.743
C03460=1175.148,138.911,-54.763,-178.545,6.436,148.744
C03461=1175.153,138.662,-54.742,-178.548,6.434,148.744
C03462=1175.157,138.413,-54.722,-178.550,6.433,148.744
C03463=1175.163,138.163,-54.702,-178.553,6.431,148.745
C03464=1175.167,137.914,-54.681,-178.556,6.429,148.745
C03465=1175.171,137.666,-54.661,-178.558,6.428,148.746
C03466=1175.177,137.417,-54.640,-178.561,6.427,148.746
C03467=1175.182,137.168,-54.620,-178.564,6.425,148.747
C03468=1175.186,136.918,-54.600,-178.566,6.423,148.747
C03469=1175.191,136.670,-54.580,-178.569,6.422,148.747
C03470=1175.196,136.420,-54.559,-178.572,6.420,148.748
C03471=1175.201,136.171,-54.539,-178.574,6.418,148.748
C03472=1175.205,135.922,-54.519,-178.577,6.417,148.749
C03473=1175.210,135.673,-54.499,-178.580,6.416,148.749
C03474=1175.215,135.424,-54.478,-178.582,6.414,148.750
C03475=1175.220,135.174,-54.458,-178.585,6.412,148.750
C03476=1175.225,134.926,-54.438,-178.588,6.411,148.750
C03477=1175.229,134.677,-54.418,-178.591,6.409,148.751
C03478=1175.234,134.427,-54.398,-178.593,6.408,148.751
C03479=1175.239,134.178,-54.377,-178.596,6.406,148.752
C03480=1175.244,133.928,-54.357,-178.599,6.405,148.752
C03481=1175.248,133.679,-54.337,-178.601,6.403,148.753
C03482=1175.253,133.430,-54.317,-178.604,6.401,148.753
C03483=1175.257,133.181,-54.297,-178.606,6.400,148.753
C03484=1175.262,132.933,-54.277,-178.609,6.399,148.754
C03485=1175.268,132.664,-54.255,-178.612,6.397,148.754
C03486=1175.273,132.396,-54.234,-178.615,6.395,148.755
C03487=1175.278,132.127,-54.212,-178.618,6.394,148.755
C03488=1175.283,131.858,-54.191,-178.621,6.392,148.756
C03489=1175.288,131.609,-54.170,-178.623,6.391,148.756
C03490=1175.292,131.360,-54.151,-178.626,6.389,148.757
C03491=1175.298,131.110,-54.130,-178.629,6.387,148.757
C03492=1175.302,130.861,-54.110,-178.632,6.386,148.758
C03493=1175.307,130.612,-54.090,-178.635,6.384,148.758
C03494=1175.312,130.363,-54.070,-178.637,6.383,148.758
C03495=1175.317,130.114,-54.050,-178.639,6.381,148.759
C03496=1175.321,129.864,-54.030,-178.642,6.380,148.759
C03497=1175.326,129.615,-54.010,-178.645,6.378,148.760
C03498=1175.331,129.367,-53.991,-178.648,6.376,148.760
C03499=1175.336,129.117,-53.971,-178.650,6.376,148.761
C03500=1175.340,128.868,-53.951,-178.653,6.374,148.761
C03501=1175.345,128.618,-53.931,-178.656,6.372,148.761
C03502=1175.350,128.370,-53.911,-178.659,6.371,148.762
C03503=1175.355,128.121,-53.891,-178.661,6.370,148.762
C03504=1175.359,127.871,-53.872,-178.664,6.368,148.763
C03505=1175.364,127.622,-53.851,-178.666,6.366,148.763
C03506=1175.369,127.373,-53.832,-178.669,6.365,148.764
C03507=1175.374,127.124,-53.812,-178.672,6.363,148.764
C03508=1175.378,126.875,-53.792,-178.674,6.362,148.765
C03509=1175.383,126.625,-53.772,-178.677,6.360,148.765
C03510=1175.389,126.376,-53.753,-178.680,6.359,148.765
C03511=1175.393,126.127,-53.733,-178.683,6.357,148.766
C03512=1175.398,125.878,-53.713,-178.685,6.356,148.766
C03513=1175.402,125.628,-53.693,-178.688,6.355,148.767
C03514=1175.408,125.379,-53.674,-178.690,6.353,148.767
C03515=1175.412,125.130,-53.654,-178.693,6.351,148.768
C03516=1175.417,124.881,-53.634,-178.696,6.350,148.768
C03517=1175.422,124.632,-53.615,-178.698,6.349,148.769
C03518=1175.426,124.383,-53.596,-178.701,6.347,148.769
C03519=1175.431,124.134,-53.575,-178.704,6.345,148.769
C03520=1175.436,123.885,-53.556,-178.707,6.344,148.770
C03521=1175.441,123.635,-53.536,-178.709,6.343,148.770
C03522=1175.446,123.386,-53.517,-178.712,6.341,148.771
C03523=1175.451,123.137,-53.497,-178.715,6.340,148.771
C03524=1175.456,122.887,-53.478,-178.717,6.338,148.772
C03525=1175.459,122.639,-53.458,-178.720,6.337,148.772
C03526=1175.465,122.390,-53.439,-178.723,6.336,148.773
C03527=1175.469,122.140,-53.419,-178.725,6.334,148.773
C03528=1175.474,121.891,-53.399,-178.728,6.332,148.773
C03529=1175.480,121.642,-53.380,-178.731,6.332,148.774
C03530=1175.484,121.392,-53.360,-178.733,6.330,148.774
C03531=1175.488,121.143,-53.341,-178.736,6.328,148.775
C03532=1175.494,120.894,-53.322,-178.739,6.326,148.775
C03533=1175.498,120.645,-53.302,-178.741,6.326,148.776
C03534=1175.504,120.396,-53.283,-178.744,6.324,148.776
C03535=1175.508,120.146,-53.264,-178.747,6.322,148.777
C03536=1175.512,119.897,-53.244,-178.749,6.321,148.777
C03537=1175.518,119.649,-53.224,-178.752,6.320,148.778
C03538=1175.522,119.399,-53.205,-178.755,6.318,148.778
C03539=1175.528,119.150,-53.186,-178.757,6.317,148.779
C03540=1175.532,118.901,-53.166,-178.760,6.316,148.779
C03541=1175.537,118.651,-53.148,-178.763,6.314,148.780
C03542=1175.542,118.402,-53.128,-178.765,6.313,148.780
C03543=1175.546,118.153,-53.109,-178.768,6.311,148.780
C03544=1175.551,117.904,-53.090,-178.771,6.310,148.781
C03545=1175.556,117.654,-53.070,-178.773,6.309,148.781
C03546=1175.561,117.405,-53.051,-178.776,6.307,148.782
C03547=1175.565,117.156,-53.032,-178.778,6.306,148.782
C03548=1175.571,116.907,-53.013,-178.782,6.305,148.783
C03549=1175.576,116.658,-52.993,-178.784,6.303,148.783
C03550=1175.580,116.408,-52.974,-178.787,6.301,148.784
C03551=1175.585,116.160,-52.955,-178.789,6.300,148.784
C03552=1175.590,115.910,-52.935,-178.792,6.299,148.785
C03553=1175.595,115.661,-52.917,-178.795,6.297,148.785
C03554=1175.599,115.411,-52.897,-178.797,6.296,148.786
C03555=1175.605,115.162,-52.878,-178.800,6.295,148.786
C03556=1175.609,114.913,-52.859,-178.803,6.293,148.787
C03557=1175.614,114.664,-52.840,-178.806,6.291,148.787
C03558=1175.619,114.415,-52.820,-178.808,6.290,148.787
C03559=1175.624,114.165,-52.802,-178.811,6.289,148.788
C03560=1175.628,113.916,-52.782,-178.814,6.287,148.788
C03561=1175.633,113.667,-52.764,-178.816,6.286,148.789
C03562=1175.638,113.418,-52.744,-178.819,6.285,148.789
C03563=1175.643,113.168,-52.725,-178.822,6.283,148.790
C03564=1175.647,112.919,-52.706,-178.824,6.282,148.790
C03565=1175.653,112.670,-52.687,-178.827,6.281,148.791
C03566=1175.657,112.421,-52.668,-178.830,6.279,148.791
C03567=1175.662,112.171,-52.649,-178.832,6.278,148.792
C03568=1175.667,111.923,-52.631,-178.835,6.277,148.792
C03569=1175.672,111.673,-52.611,-178.838,6.275,148.793
C03570=1175.677,111.424,-52.593,-178.840,6.274,148.793
C03571=1175.681,111.175,-52.573,-178.843,6.273,148.794
C03572=1175.687,110.926,-52.554,-178.846,6.271,148.794
C03573=1175.691,110.676,-52.536,-178.848,6.270,148.795
C03574=1175.696,110.427,-52.517,-178.851,6.269,148.795
C03575=1175.701,110.178,-52.498,-178.853,6.267,148.795
C03576=1175.706,109.928,-52.479,-178.856,6.266,148.796
C03577=1175.711,109.680,-52.460,-178.859,6.265,148.796
C03578=1175.715,109.430,-52.442,-178.861,6.263,148.797
C03579=1175.720,109.181,-52.423,-178.864,6.262,148.798
C03580=1175.724,108.932,-52.403,-178.867,6.261,148.798
C03581=1175.730,108.682,-52.385,-178.869,6.259,148.798
C03582=1175.735,108.434,-52.366,-178.872,6.258,148.799
C03583=1175.740,108.183,-52.347,-178.875,6.257,148.799
C03584=1175.744,107.935,-52.329,-178.878,6.255,148.800
C03585=1175.749,107.685,-52.310,-178.880,6.254,148.800
C03586=1175.754,107.436,-52.291,-178.883,6.253,148.801
C03587=1175.759,107.187,-52.273,-178.886,6.251,148.801
C03588=1175.764,106.937,-52.253,-178.888,6.250,148.802
C03589=1175.769,106.669,-52.234,-178.891,6.249,148.802
C03590=1175.774,106.401,-52.213,-178.894,6.247,148.803
C03591=1175.779,106.132,-52.193,-178.897,6.245,148.803
C03592=1175.784,105.864,-52.173,-178.900,6.244,148.804
C03593=1175.789,105.615,-52.155,-178.902,6.243,148.804
C03594=1175.795,105.366,-52.136,-178.905,6.241,148.805
C03595=1175.799,105.116,-52.117,-178.908,6.240,148.805
C03596=1175.804,104.867,-52.098,-178.910,6.239,148.806
C03597=1175.809,104.618,-52.081,-178.913,6.237,148.806
C03598=1175.813,104.368,-52.061,-178.916,6.237,148.807
C03599=1175.819,104.119,-52.043,-178.918,6.235,148.807
C03600=1175.824,103.870,-52.024,-178.921,6.233,148.808
C03601=1175.828,103.621,-52.006,-178.924,6.233,148.808
C03602=1175.833,103.371,-51.988,-178.926,6.231,148.809
C03603=1175.838,103.122,-51.969,-178.929,6.229,148.809
C03604=1175.842,102.873,-51.950,-178.932,6.229,148.810
C03605=1175.847,102.623,-51.932,-178.934,6.227,148.810
C03606=1175.853,102.375,-51.913,-178.936,6.226,148.811
C03607=1175.858,102.125,-51.895,-178.940,6.225,148.811
C03608=1175.862,101.875,-51.877,-178.942,6.223,148.812
C03609=1175.866,101.627,-51.858,-178.945,6.223,148.812
C03610=1175.872,101.377,-51.839,-178.948,6.221,148.813
C03611=1175.876,101.128,-51.821,-178.950,6.220,148.813
C03612=1175.881,100.878,-51.803,-178.953,6.219,148.814
C03613=1175.886,100.630,-51.784,-178.956,6.217,148.814
C03614=1175.892,100.380,-51.766,-178.958,6.216,148.815
C03615=1175.896,100.130,-51.747,-178.961,6.215,148.815
C03616=1175.901,99.881,-51.729,-178.963,6.214,148.816
C03617=1175.906,99.632,-51.711,-178.966,6.212,148.816
C03618=1175.910,99.384,-51.693,-178.969,6.211,148.817
C03619=1175.915,99.133,-51.674,-178.971,6.210,148.817
C03620=1175.920,98.884,-51.656,-178.974,6.208,148.818
C03621=1175.925,98.635,-51.638,-178.977,6.208,148.818
C03622=1175.930,98.386,-51.620,-178.979,6.206,148.819
C03623=1175.935,98.137,-51.602,-178.983,6.204,148.819
C03624=1175.939,97.887,-51.583,-178.985,6.204,148.820
C03625=1175.945,97.638,-51.564,-178.987,6.202,148.820
C03626=1175.950,97.389,-51.546,-178.990,6.201,148.821
C03627=1175.955,97.140,-51.528,-178.993,6.200,148.821
C03628=1175.959,96.890,-51.510,-178.995,6.198,148.822
C03629=1175.964,96.641,-51.492,-178.998,6.197,148.822
C03630=1175.969,96.391,-51.474,-179.001,6.196,148.823
C03631=1175.974,96.142,-51.456,-179.003,6.195,148.823
C03632=1175.978,95.893,-51.438,-179.006,6.193,148.824
C03633=1175.984,95.644,-51.419,-179.008,6.192,148.824
C03634=1175.989,95.394,-51.401,-179.011,6.191,148.825
C03635=1175.993,95.144,-51.383,-179.014,6.189,148.825
C03636=1175.998,94.895,-51.365,-179.017,6.189,148.826
C03637=1176.003,94.646,-51.347,-179.019,6.187,148.826
C03638=1176.008,94.397,-51.329,-179.022,6.186,148.827
C03639=1176.013,94.148,-51.311,-179.025,6.185,148.827
C03640=1176.018,93.899,-51.293,-179.027,6.184,148.828
C03641=1176.023,93.649,-51.275,-179.030,6.183,148.828
C03642=1176.027,93.400,-51.257,-179.032,6.182,148.829
C03643=1176.032,93.150,-51.239,-179.035,6.180,148.829
C03644=1176.037,92.901,-51.221,-179.038,6.179,148.830
